(* Logix 5000 project; controller reports 1756-L63 rev 20.11; software revision 20.04; part 18 of 52 *)

        [994].time.Day := 13, [994].time.Hour := 3, [994].time.Minute := 14, [994].time.Second := 59, [995].log_data[0].min := 1.0, [995].log_data[0].max := 1.0, [995].log_data[0].total := 300.0, [995].log_data[0].time := 300.0, [995].log_data[0].minminute := 15, [995].log_data[0].maxminute := 15, [995].log_data[0].valid := 1, [995].log_data[1].valid := 1, [995].log_data[2].valid := 1, [995].log_data[3].valid := 1, [995].log_data[4].valid := 1, [995].log_data[5].valid := 1, [995].log_data[6].valid := 1, [995].log_data[7].valid := 1, [995].log_data[8].valid := 1, [995].log_data[9].valid := 1, [995].log_data[10].valid := 1, [995].log_data[11].valid := 1, [995].log_data[12].valid := 1, [995].log_data[13].valid := 1, [995].log_data[14].valid := 1, [995].log_data[15].valid := 1, [995].log_data[16].valid := 1, [995].log_data[17].valid := 1, [995].log_data[18].valid := 1, [995].log_data[19].valid := 1, [995].time.Year := 2023, [995].time.Month := 1, [995].time.Day := 13, [995].time.Hour := 3, [995].time.Minute := 19, [995].time.Second := 59, [996].log_data[0].min := 1.0, [996].log_data[0].max := 1.0, [996].log_data[0].total := 300.0, [996].log_data[0].time := 300.0, [996].log_data[0].minminute := 20, [996].log_data[0].maxminute := 20, [996].log_data[0].valid := 1, [996].log_data[1].valid := 1, [996].log_data[2].valid := 1, [996].log_data[3].valid := 1, [996].log_data[4].valid := 1, [996].log_data[5].valid := 1, [996].log_data[6].valid := 1, [996].log_data[7].valid := 1, [996].log_data[8].valid := 1, [996].log_data[9].valid := 1, [996].log_data[10].valid := 1, [996].log_data[11].valid := 1, [996].log_data[12].valid := 1, [996].log_data[13].valid := 1, [996].log_data[14].valid := 1, [996].log_data[15].valid := 1, [996].log_data[16].valid := 1, [996].log_data[17].valid := 1,
        [996].log_data[18].valid := 1, [996].log_data[19].valid := 1, [996].time.Year := 2023, [996].time.Month := 1, [996].time.Day := 13, [996].time.Hour := 3, [996].time.Minute := 24, [996].time.Second := 59, [997].log_data[0].min := 1.0, [997].log_data[0].max := 1.0, [997].log_data[0].total := 300.0, [997].log_data[0].time := 300.0, [997].log_data[0].minminute := 25, [997].log_data[0].maxminute := 25, [997].log_data[0].valid := 1, [997].log_data[1].valid := 1, [997].log_data[2].valid := 1, [997].log_data[3].valid := 1, [997].log_data[4].valid := 1, [997].log_data[5].valid := 1, [997].log_data[6].valid := 1, [997].log_data[7].valid := 1, [997].log_data[8].valid := 1, [997].log_data[9].valid := 1, [997].log_data[10].valid := 1, [997].log_data[11].valid := 1, [997].log_data[12].valid := 1, [997].log_data[13].valid := 1, [997].log_data[14].valid := 1, [997].log_data[15].valid := 1, [997].log_data[16].valid := 1, [997].log_data[17].valid := 1, [997].log_data[18].valid := 1, [997].log_data[19].valid := 1, [997].time.Year := 2023, [997].time.Month := 1, [997].time.Day := 13, [997].time.Hour := 3, [997].time.Minute := 29, [997].time.Second := 59, [998].log_data[0].min := 1.0, [998].log_data[0].max := 1.0, [998].log_data[0].total := 300.0, [998].log_data[0].time := 300.0, [998].log_data[0].minminute := 30, [998].log_data[0].maxminute := 30, [998].log_data[0].valid := 1, [998].log_data[1].valid := 1, [998].log_data[2].valid := 1, [998].log_data[3].valid := 1, [998].log_data[4].valid := 1, [998].log_data[5].valid := 1, [998].log_data[6].valid := 1, [998].log_data[7].valid := 1, [998].log_data[8].valid := 1, [998].log_data[9].valid := 1, [998].log_data[10].valid := 1, [998].log_data[11].valid := 1, [998].log_data[12].valid := 1, [998].log_data[13].valid := 1,
        [998].log_data[14].valid := 1, [998].log_data[15].valid := 1, [998].log_data[16].valid := 1, [998].log_data[17].valid := 1, [998].log_data[18].valid := 1, [998].log_data[19].valid := 1, [998].time.Year := 2023, [998].time.Month := 1, [998].time.Day := 13, [998].time.Hour := 3, [998].time.Minute := 34, [998].time.Second := 59, [999].log_data[0].min := 1.0, [999].log_data[0].max := 1.0, [999].log_data[0].total := 300.0, [999].log_data[0].time := 300.0, [999].log_data[0].minminute := 35, [999].log_data[0].maxminute := 35, [999].log_data[0].valid := 1, [999].log_data[1].valid := 1, [999].log_data[2].valid := 1, [999].log_data[3].valid := 1, [999].log_data[4].valid := 1, [999].log_data[5].valid := 1, [999].log_data[6].valid := 1, [999].log_data[7].valid := 1, [999].log_data[8].valid := 1, [999].log_data[9].valid := 1, [999].log_data[10].valid := 1, [999].log_data[11].valid := 1, [999].log_data[12].valid := 1, [999].log_data[13].valid := 1, [999].log_data[14].valid := 1, [999].log_data[15].valid := 1, [999].log_data[16].valid := 1, [999].log_data[17].valid := 1, [999].log_data[18].valid := 1, [999].log_data[19].valid := 1, [999].time.Year := 2023, [999].time.Month := 1, [999].time.Day := 13, [999].time.Hour := 3, [999].time.Minute := 39, [999].time.Second := 59, [1000].log_data[0].min := 1.0, [1000].log_data[0].max := 1.0, [1000].log_data[0].total := 300.0, [1000].log_data[0].time := 300.0, [1000].log_data[0].minminute := 40, [1000].log_data[0].maxminute := 40, [1000].log_data[0].valid := 1, [1000].log_data[1].valid := 1, [1000].log_data[2].valid := 1, [1000].log_data[3].valid := 1, [1000].log_data[4].valid := 1, [1000].log_data[5].valid := 1, [1000].log_data[6].valid := 1, [1000].log_data[7].valid := 1, [1000].log_data[8].valid := 1, [1000].log_data[9].valid := 1,
        [1000].log_data[10].valid := 1, [1000].log_data[11].valid := 1, [1000].log_data[12].valid := 1, [1000].log_data[13].valid := 1, [1000].log_data[14].valid := 1, [1000].log_data[15].valid := 1, [1000].log_data[16].valid := 1, [1000].log_data[17].valid := 1, [1000].log_data[18].valid := 1, [1000].log_data[19].valid := 1, [1000].time.Year := 2023, [1000].time.Month := 1, [1000].time.Day := 13, [1000].time.Hour := 3, [1000].time.Minute := 44, [1000].time.Second := 59, [1001].log_data[0].min := 1.0, [1001].log_data[0].max := 1.0, [1001].log_data[0].total := 300.0, [1001].log_data[0].time := 300.0, [1001].log_data[0].minminute := 45, [1001].log_data[0].maxminute := 45, [1001].log_data[0].valid := 1, [1001].log_data[1].valid := 1, [1001].log_data[2].valid := 1, [1001].log_data[3].valid := 1, [1001].log_data[4].valid := 1, [1001].log_data[5].valid := 1, [1001].log_data[6].valid := 1, [1001].log_data[7].valid := 1, [1001].log_data[8].valid := 1, [1001].log_data[9].valid := 1, [1001].log_data[10].valid := 1, [1001].log_data[11].valid := 1, [1001].log_data[12].valid := 1, [1001].log_data[13].valid := 1, [1001].log_data[14].valid := 1, [1001].log_data[15].valid := 1, [1001].log_data[16].valid := 1, [1001].log_data[17].valid := 1, [1001].log_data[18].valid := 1, [1001].log_data[19].valid := 1, [1001].time.Year := 2023, [1001].time.Month := 1, [1001].time.Day := 13, [1001].time.Hour := 3, [1001].time.Minute := 49, [1001].time.Second := 59, [1002].log_data[0].min := 1.0, [1002].log_data[0].max := 1.0, [1002].log_data[0].total := 300.0, [1002].log_data[0].time := 300.0, [1002].log_data[0].minminute := 50, [1002].log_data[0].maxminute := 50, [1002].log_data[0].valid := 1, [1002].log_data[1].valid := 1, [1002].log_data[2].valid := 1, [1002].log_data[3].valid := 1, [1002].log_data[4].valid := 1, [1002].log_data[5].valid := 1,
        [1002].log_data[6].valid := 1, [1002].log_data[7].valid := 1, [1002].log_data[8].valid := 1, [1002].log_data[9].valid := 1, [1002].log_data[10].valid := 1, [1002].log_data[11].valid := 1, [1002].log_data[12].valid := 1, [1002].log_data[13].valid := 1, [1002].log_data[14].valid := 1, [1002].log_data[15].valid := 1, [1002].log_data[16].valid := 1, [1002].log_data[17].valid := 1, [1002].log_data[18].valid := 1, [1002].log_data[19].valid := 1, [1002].time.Year := 2023, [1002].time.Month := 1, [1002].time.Day := 13, [1002].time.Hour := 3, [1002].time.Minute := 54, [1002].time.Second := 59, [1003].log_data[0].min := 1.0, [1003].log_data[0].max := 1.0, [1003].log_data[0].total := 300.0, [1003].log_data[0].time := 300.0, [1003].log_data[0].minminute := 55, [1003].log_data[0].maxminute := 55, [1003].log_data[0].valid := 1, [1003].log_data[1].valid := 1, [1003].log_data[2].valid := 1, [1003].log_data[3].valid := 1, [1003].log_data[4].valid := 1, [1003].log_data[5].valid := 1, [1003].log_data[6].valid := 1, [1003].log_data[7].valid := 1, [1003].log_data[8].valid := 1, [1003].log_data[9].valid := 1, [1003].log_data[10].valid := 1, [1003].log_data[11].valid := 1, [1003].log_data[12].valid := 1, [1003].log_data[13].valid := 1, [1003].log_data[14].valid := 1, [1003].log_data[15].valid := 1, [1003].log_data[16].valid := 1, [1003].log_data[17].valid := 1, [1003].log_data[18].valid := 1, [1003].log_data[19].valid := 1, [1003].time.Year := 2023, [1003].time.Month := 1, [1003].time.Day := 13, [1003].time.Hour := 3, [1003].time.Minute := 59, [1003].time.Second := 59, [1004].log_data[0].min := 1.0, [1004].log_data[0].max := 1.0, [1004].log_data[0].total := 300.0, [1004].log_data[0].time := 300.0, [1004].log_data[0].valid := 1, [1004].log_data[1].valid := 1, [1004].log_data[2].valid := 1, [1004].log_data[3].valid := 1,
        [1004].log_data[4].valid := 1, [1004].log_data[5].valid := 1, [1004].log_data[6].valid := 1, [1004].log_data[7].valid := 1, [1004].log_data[8].valid := 1, [1004].log_data[9].valid := 1, [1004].log_data[10].valid := 1, [1004].log_data[11].valid := 1, [1004].log_data[12].valid := 1, [1004].log_data[13].valid := 1, [1004].log_data[14].valid := 1, [1004].log_data[15].valid := 1, [1004].log_data[16].valid := 1, [1004].log_data[17].valid := 1, [1004].log_data[18].valid := 1, [1004].log_data[19].valid := 1, [1004].time.Year := 2023, [1004].time.Month := 1, [1004].time.Day := 13, [1004].time.Hour := 4, [1004].time.Minute := 4, [1004].time.Second := 59, [1005].log_data[0].min := 1.0, [1005].log_data[0].max := 1.0, [1005].log_data[0].total := 300.0, [1005].log_data[0].time := 300.0, [1005].log_data[0].minminute := 5, [1005].log_data[0].maxminute := 5, [1005].log_data[0].valid := 1, [1005].log_data[1].valid := 1, [1005].log_data[2].valid := 1, [1005].log_data[3].valid := 1, [1005].log_data[4].valid := 1, [1005].log_data[5].valid := 1, [1005].log_data[6].valid := 1, [1005].log_data[7].valid := 1, [1005].log_data[8].valid := 1, [1005].log_data[9].valid := 1, [1005].log_data[10].valid := 1, [1005].log_data[11].valid := 1, [1005].log_data[12].valid := 1, [1005].log_data[13].valid := 1, [1005].log_data[14].valid := 1, [1005].log_data[15].valid := 1, [1005].log_data[16].valid := 1, [1005].log_data[17].valid := 1, [1005].log_data[18].valid := 1, [1005].log_data[19].valid := 1, [1005].time.Year := 2023, [1005].time.Month := 1, [1005].time.Day := 13, [1005].time.Hour := 4, [1005].time.Minute := 9, [1005].time.Second := 59, [1006].log_data[0].min := 1.0, [1006].log_data[0].max := 1.0, [1006].log_data[0].total := 300.0, [1006].log_data[0].time := 300.0, [1006].log_data[0].minminute := 10, [1006].log_data[0].maxminute := 10,
        [1006].log_data[0].valid := 1, [1006].log_data[1].valid := 1, [1006].log_data[2].valid := 1, [1006].log_data[3].valid := 1, [1006].log_data[4].valid := 1, [1006].log_data[5].valid := 1, [1006].log_data[6].valid := 1, [1006].log_data[7].valid := 1, [1006].log_data[8].valid := 1, [1006].log_data[9].valid := 1, [1006].log_data[10].valid := 1, [1006].log_data[11].valid := 1, [1006].log_data[12].valid := 1, [1006].log_data[13].valid := 1, [1006].log_data[14].valid := 1, [1006].log_data[15].valid := 1, [1006].log_data[16].valid := 1, [1006].log_data[17].valid := 1, [1006].log_data[18].valid := 1, [1006].log_data[19].valid := 1, [1006].time.Year := 2023, [1006].time.Month := 1, [1006].time.Day := 13, [1006].time.Hour := 4, [1006].time.Minute := 14, [1006].time.Second := 59, [1007].log_data[0].min := 1.0, [1007].log_data[0].max := 1.0, [1007].log_data[0].total := 300.0, [1007].log_data[0].time := 300.0, [1007].log_data[0].minminute := 15, [1007].log_data[0].maxminute := 15, [1007].log_data[0].valid := 1, [1007].log_data[1].valid := 1, [1007].log_data[2].valid := 1, [1007].log_data[3].valid := 1, [1007].log_data[4].valid := 1, [1007].log_data[5].valid := 1, [1007].log_data[6].valid := 1, [1007].log_data[7].valid := 1, [1007].log_data[8].valid := 1, [1007].log_data[9].valid := 1, [1007].log_data[10].valid := 1, [1007].log_data[11].valid := 1, [1007].log_data[12].valid := 1, [1007].log_data[13].valid := 1, [1007].log_data[14].valid := 1, [1007].log_data[15].valid := 1, [1007].log_data[16].valid := 1, [1007].log_data[17].valid := 1, [1007].log_data[18].valid := 1, [1007].log_data[19].valid := 1, [1007].time.Year := 2023, [1007].time.Month := 1, [1007].time.Day := 13, [1007].time.Hour := 4, [1007].time.Minute := 19, [1007].time.Second := 59, [1008].log_data[0].min := 1.0, [1008].log_data[0].max := 1.0,
        [1008].log_data[0].total := 300.0, [1008].log_data[0].time := 300.0, [1008].log_data[0].minminute := 20, [1008].log_data[0].maxminute := 20, [1008].log_data[0].valid := 1, [1008].log_data[1].valid := 1, [1008].log_data[2].valid := 1, [1008].log_data[3].valid := 1, [1008].log_data[4].valid := 1, [1008].log_data[5].valid := 1, [1008].log_data[6].valid := 1, [1008].log_data[7].valid := 1, [1008].log_data[8].valid := 1, [1008].log_data[9].valid := 1, [1008].log_data[10].valid := 1, [1008].log_data[11].valid := 1, [1008].log_data[12].valid := 1, [1008].log_data[13].valid := 1, [1008].log_data[14].valid := 1, [1008].log_data[15].valid := 1, [1008].log_data[16].valid := 1, [1008].log_data[17].valid := 1, [1008].log_data[18].valid := 1, [1008].log_data[19].valid := 1, [1008].time.Year := 2023, [1008].time.Month := 1, [1008].time.Day := 13, [1008].time.Hour := 4, [1008].time.Minute := 24, [1008].time.Second := 59, [1009].log_data[0].min := 1.0, [1009].log_data[0].max := 1.0, [1009].log_data[0].total := 300.0, [1009].log_data[0].time := 300.0, [1009].log_data[0].minminute := 25, [1009].log_data[0].maxminute := 25, [1009].log_data[0].valid := 1, [1009].log_data[1].valid := 1, [1009].log_data[2].valid := 1, [1009].log_data[3].valid := 1, [1009].log_data[4].valid := 1, [1009].log_data[5].valid := 1, [1009].log_data[6].valid := 1, [1009].log_data[7].valid := 1, [1009].log_data[8].valid := 1, [1009].log_data[9].valid := 1, [1009].log_data[10].valid := 1, [1009].log_data[11].valid := 1, [1009].log_data[12].valid := 1, [1009].log_data[13].valid := 1, [1009].log_data[14].valid := 1, [1009].log_data[15].valid := 1, [1009].log_data[16].valid := 1, [1009].log_data[17].valid := 1, [1009].log_data[18].valid := 1, [1009].log_data[19].valid := 1, [1009].time.Year := 2023, [1009].time.Month := 1, [1009].time.Day := 13, [1009].time.Hour := 4,
        [1009].time.Minute := 29, [1009].time.Second := 59, [1010].log_data[0].min := 1.0, [1010].log_data[0].max := 1.0, [1010].log_data[0].total := 300.0, [1010].log_data[0].time := 300.0, [1010].log_data[0].minminute := 30, [1010].log_data[0].maxminute := 30, [1010].log_data[0].valid := 1, [1010].log_data[1].valid := 1, [1010].log_data[2].valid := 1, [1010].log_data[3].valid := 1, [1010].log_data[4].valid := 1, [1010].log_data[5].valid := 1, [1010].log_data[6].valid := 1, [1010].log_data[7].valid := 1, [1010].log_data[8].valid := 1, [1010].log_data[9].valid := 1, [1010].log_data[10].valid := 1, [1010].log_data[11].valid := 1, [1010].log_data[12].valid := 1, [1010].log_data[13].valid := 1, [1010].log_data[14].valid := 1, [1010].log_data[15].valid := 1, [1010].log_data[16].valid := 1, [1010].log_data[17].valid := 1, [1010].log_data[18].valid := 1, [1010].log_data[19].valid := 1, [1010].time.Year := 2023, [1010].time.Month := 1, [1010].time.Day := 13, [1010].time.Hour := 4, [1010].time.Minute := 34, [1010].time.Second := 59, [1011].log_data[0].min := 1.0, [1011].log_data[0].max := 1.0, [1011].log_data[0].total := 300.0, [1011].log_data[0].time := 300.0, [1011].log_data[0].minminute := 35, [1011].log_data[0].maxminute := 35, [1011].log_data[0].valid := 1, [1011].log_data[1].valid := 1, [1011].log_data[2].valid := 1, [1011].log_data[3].valid := 1, [1011].log_data[4].valid := 1, [1011].log_data[5].valid := 1, [1011].log_data[6].valid := 1, [1011].log_data[7].valid := 1, [1011].log_data[8].valid := 1, [1011].log_data[9].valid := 1, [1011].log_data[10].valid := 1, [1011].log_data[11].valid := 1, [1011].log_data[12].valid := 1, [1011].log_data[13].valid := 1, [1011].log_data[14].valid := 1, [1011].log_data[15].valid := 1, [1011].log_data[16].valid := 1, [1011].log_data[17].valid := 1, [1011].log_data[18].valid := 1, [1011].log_data[19].valid := 1,
        [1011].time.Year := 2023, [1011].time.Month := 1, [1011].time.Day := 13, [1011].time.Hour := 4, [1011].time.Minute := 39, [1011].time.Second := 59, [1012].log_data[0].min := 1.0, [1012].log_data[0].max := 1.0, [1012].log_data[0].total := 300.0, [1012].log_data[0].time := 300.0, [1012].log_data[0].minminute := 40, [1012].log_data[0].maxminute := 40, [1012].log_data[0].valid := 1, [1012].log_data[1].valid := 1, [1012].log_data[2].valid := 1, [1012].log_data[3].valid := 1, [1012].log_data[4].valid := 1, [1012].log_data[5].valid := 1, [1012].log_data[6].valid := 1, [1012].log_data[7].valid := 1, [1012].log_data[8].valid := 1, [1012].log_data[9].valid := 1, [1012].log_data[10].valid := 1, [1012].log_data[11].valid := 1, [1012].log_data[12].valid := 1, [1012].log_data[13].valid := 1, [1012].log_data[14].valid := 1, [1012].log_data[15].valid := 1, [1012].log_data[16].valid := 1, [1012].log_data[17].valid := 1, [1012].log_data[18].valid := 1, [1012].log_data[19].valid := 1, [1012].time.Year := 2023, [1012].time.Month := 1, [1012].time.Day := 13, [1012].time.Hour := 4, [1012].time.Minute := 44, [1012].time.Second := 59, [1013].log_data[0].min := 1.0, [1013].log_data[0].max := 1.0, [1013].log_data[0].total := 300.0, [1013].log_data[0].time := 300.0, [1013].log_data[0].minminute := 45, [1013].log_data[0].maxminute := 45, [1013].log_data[0].valid := 1, [1013].log_data[1].valid := 1, [1013].log_data[2].valid := 1, [1013].log_data[3].valid := 1, [1013].log_data[4].valid := 1, [1013].log_data[5].valid := 1, [1013].log_data[6].valid := 1, [1013].log_data[7].valid := 1, [1013].log_data[8].valid := 1, [1013].log_data[9].valid := 1, [1013].log_data[10].valid := 1, [1013].log_data[11].valid := 1, [1013].log_data[12].valid := 1, [1013].log_data[13].valid := 1, [1013].log_data[14].valid := 1, [1013].log_data[15].valid := 1,
        [1013].log_data[16].valid := 1, [1013].log_data[17].valid := 1, [1013].log_data[18].valid := 1, [1013].log_data[19].valid := 1, [1013].time.Year := 2023, [1013].time.Month := 1, [1013].time.Day := 13, [1013].time.Hour := 4, [1013].time.Minute := 49, [1013].time.Second := 59, [1014].log_data[0].min := 1.0, [1014].log_data[0].max := 1.0, [1014].log_data[0].total := 300.0, [1014].log_data[0].time := 300.0, [1014].log_data[0].minminute := 50, [1014].log_data[0].maxminute := 50, [1014].log_data[0].valid := 1, [1014].log_data[1].valid := 1, [1014].log_data[2].valid := 1, [1014].log_data[3].valid := 1, [1014].log_data[4].valid := 1, [1014].log_data[5].valid := 1, [1014].log_data[6].valid := 1, [1014].log_data[7].valid := 1, [1014].log_data[8].valid := 1, [1014].log_data[9].valid := 1, [1014].log_data[10].valid := 1, [1014].log_data[11].valid := 1, [1014].log_data[12].valid := 1, [1014].log_data[13].valid := 1, [1014].log_data[14].valid := 1, [1014].log_data[15].valid := 1, [1014].log_data[16].valid := 1, [1014].log_data[17].valid := 1, [1014].log_data[18].valid := 1, [1014].log_data[19].valid := 1, [1014].time.Year := 2023, [1014].time.Month := 1, [1014].time.Day := 13, [1014].time.Hour := 4, [1014].time.Minute := 54, [1014].time.Second := 59, [1015].log_data[0].min := 1.0, [1015].log_data[0].max := 1.0, [1015].log_data[0].total := 300.0, [1015].log_data[0].time := 300.0, [1015].log_data[0].minminute := 55, [1015].log_data[0].maxminute := 55, [1015].log_data[0].valid := 1, [1015].log_data[1].valid := 1, [1015].log_data[2].valid := 1, [1015].log_data[3].valid := 1, [1015].log_data[4].valid := 1, [1015].log_data[5].valid := 1, [1015].log_data[6].valid := 1, [1015].log_data[7].valid := 1, [1015].log_data[8].valid := 1, [1015].log_data[9].valid := 1, [1015].log_data[10].valid := 1, [1015].log_data[11].valid := 1,
        [1015].log_data[12].valid := 1, [1015].log_data[13].valid := 1, [1015].log_data[14].valid := 1, [1015].log_data[15].valid := 1, [1015].log_data[16].valid := 1, [1015].log_data[17].valid := 1, [1015].log_data[18].valid := 1, [1015].log_data[19].valid := 1, [1015].time.Year := 2023, [1015].time.Month := 1, [1015].time.Day := 13, [1015].time.Hour := 4, [1015].time.Minute := 59, [1015].time.Second := 59, [1016].log_data[0].min := 1.0, [1016].log_data[0].max := 1.0, [1016].log_data[0].total := 300.0, [1016].log_data[0].time := 300.0, [1016].log_data[0].valid := 1, [1016].log_data[1].valid := 1, [1016].log_data[2].valid := 1, [1016].log_data[3].valid := 1, [1016].log_data[4].valid := 1, [1016].log_data[5].valid := 1, [1016].log_data[6].valid := 1, [1016].log_data[7].valid := 1, [1016].log_data[8].valid := 1, [1016].log_data[9].valid := 1, [1016].log_data[10].valid := 1, [1016].log_data[11].valid := 1, [1016].log_data[12].valid := 1, [1016].log_data[13].valid := 1, [1016].log_data[14].valid := 1, [1016].log_data[15].valid := 1, [1016].log_data[16].valid := 1, [1016].log_data[17].valid := 1, [1016].log_data[18].valid := 1, [1016].log_data[19].valid := 1, [1016].time.Year := 2023, [1016].time.Month := 1, [1016].time.Day := 13, [1016].time.Hour := 5, [1016].time.Minute := 4, [1016].time.Second := 59, [1017].log_data[0].min := 1.0, [1017].log_data[0].max := 1.0, [1017].log_data[0].total := 300.0, [1017].log_data[0].time := 300.0, [1017].log_data[0].minminute := 5, [1017].log_data[0].maxminute := 5, [1017].log_data[0].valid := 1, [1017].log_data[1].valid := 1, [1017].log_data[2].valid := 1, [1017].log_data[3].valid := 1, [1017].log_data[4].valid := 1, [1017].log_data[5].valid := 1, [1017].log_data[6].valid := 1, [1017].log_data[7].valid := 1, [1017].log_data[8].valid := 1, [1017].log_data[9].valid := 1,
        [1017].log_data[10].valid := 1, [1017].log_data[11].valid := 1, [1017].log_data[12].valid := 1, [1017].log_data[13].valid := 1, [1017].log_data[14].valid := 1, [1017].log_data[15].valid := 1, [1017].log_data[16].valid := 1, [1017].log_data[17].valid := 1, [1017].log_data[18].valid := 1, [1017].log_data[19].valid := 1, [1017].time.Year := 2023, [1017].time.Month := 1, [1017].time.Day := 13, [1017].time.Hour := 5, [1017].time.Minute := 9, [1017].time.Second := 59, [1018].log_data[0].min := 1.0, [1018].log_data[0].max := 1.0, [1018].log_data[0].total := 300.0, [1018].log_data[0].time := 300.0, [1018].log_data[0].minminute := 10, [1018].log_data[0].maxminute := 10, [1018].log_data[0].valid := 1, [1018].log_data[1].valid := 1, [1018].log_data[2].valid := 1, [1018].log_data[3].valid := 1, [1018].log_data[4].valid := 1, [1018].log_data[5].valid := 1, [1018].log_data[6].valid := 1, [1018].log_data[7].valid := 1, [1018].log_data[8].valid := 1, [1018].log_data[9].valid := 1, [1018].log_data[10].valid := 1, [1018].log_data[11].valid := 1, [1018].log_data[12].valid := 1, [1018].log_data[13].valid := 1, [1018].log_data[14].valid := 1, [1018].log_data[15].valid := 1, [1018].log_data[16].valid := 1, [1018].log_data[17].valid := 1, [1018].log_data[18].valid := 1, [1018].log_data[19].valid := 1, [1018].time.Year := 2023, [1018].time.Month := 1, [1018].time.Day := 13, [1018].time.Hour := 5, [1018].time.Minute := 14, [1018].time.Second := 59, [1019].log_data[0].min := 1.0, [1019].log_data[0].max := 1.0, [1019].log_data[0].total := 300.0, [1019].log_data[0].time := 300.0, [1019].log_data[0].minminute := 15, [1019].log_data[0].maxminute := 15, [1019].log_data[0].valid := 1, [1019].log_data[1].valid := 1, [1019].log_data[2].valid := 1, [1019].log_data[3].valid := 1, [1019].log_data[4].valid := 1, [1019].log_data[5].valid := 1,
        [1019].log_data[6].valid := 1, [1019].log_data[7].valid := 1, [1019].log_data[8].valid := 1, [1019].log_data[9].valid := 1, [1019].log_data[10].valid := 1, [1019].log_data[11].valid := 1, [1019].log_data[12].valid := 1, [1019].log_data[13].valid := 1, [1019].log_data[14].valid := 1, [1019].log_data[15].valid := 1, [1019].log_data[16].valid := 1, [1019].log_data[17].valid := 1, [1019].log_data[18].valid := 1, [1019].log_data[19].valid := 1, [1019].time.Year := 2023, [1019].time.Month := 1, [1019].time.Day := 13, [1019].time.Hour := 5, [1019].time.Minute := 19, [1019].time.Second := 59, [1020].log_data[0].min := 1.0, [1020].log_data[0].max := 1.0, [1020].log_data[0].total := 300.0, [1020].log_data[0].time := 300.0, [1020].log_data[0].minminute := 20, [1020].log_data[0].maxminute := 20, [1020].log_data[0].valid := 1, [1020].log_data[1].valid := 1, [1020].log_data[2].valid := 1, [1020].log_data[3].valid := 1, [1020].log_data[4].valid := 1, [1020].log_data[5].valid := 1, [1020].log_data[6].valid := 1, [1020].log_data[7].valid := 1, [1020].log_data[8].valid := 1, [1020].log_data[9].valid := 1, [1020].log_data[10].valid := 1, [1020].log_data[11].valid := 1, [1020].log_data[12].valid := 1, [1020].log_data[13].valid := 1, [1020].log_data[14].valid := 1, [1020].log_data[15].valid := 1, [1020].log_data[16].valid := 1, [1020].log_data[17].valid := 1, [1020].log_data[18].valid := 1, [1020].log_data[19].valid := 1, [1020].time.Year := 2023, [1020].time.Month := 1, [1020].time.Day := 13, [1020].time.Hour := 5, [1020].time.Minute := 24, [1020].time.Second := 59, [1021].log_data[0].min := 1.0, [1021].log_data[0].max := 1.0, [1021].log_data[0].total := 300.0, [1021].log_data[0].time := 300.0, [1021].log_data[0].minminute := 25, [1021].log_data[0].maxminute := 25, [1021].log_data[0].valid := 1, [1021].log_data[1].valid := 1,
        [1021].log_data[2].valid := 1, [1021].log_data[3].valid := 1, [1021].log_data[4].valid := 1, [1021].log_data[5].valid := 1, [1021].log_data[6].valid := 1, [1021].log_data[7].valid := 1, [1021].log_data[8].valid := 1, [1021].log_data[9].valid := 1, [1021].log_data[10].valid := 1, [1021].log_data[11].valid := 1, [1021].log_data[12].valid := 1, [1021].log_data[13].valid := 1, [1021].log_data[14].valid := 1, [1021].log_data[15].valid := 1, [1021].log_data[16].valid := 1, [1021].log_data[17].valid := 1, [1021].log_data[18].valid := 1, [1021].log_data[19].valid := 1, [1021].time.Year := 2023, [1021].time.Month := 1, [1021].time.Day := 13, [1021].time.Hour := 5, [1021].time.Minute := 29, [1021].time.Second := 59, [1022].log_data[0].min := 1.0, [1022].log_data[0].max := 1.0, [1022].log_data[0].total := 300.0, [1022].log_data[0].time := 300.0, [1022].log_data[0].minminute := 30, [1022].log_data[0].maxminute := 30, [1022].log_data[0].valid := 1, [1022].log_data[1].valid := 1, [1022].log_data[2].valid := 1, [1022].log_data[3].valid := 1, [1022].log_data[4].valid := 1, [1022].log_data[5].valid := 1, [1022].log_data[6].valid := 1, [1022].log_data[7].valid := 1, [1022].log_data[8].valid := 1, [1022].log_data[9].valid := 1, [1022].log_data[10].valid := 1, [1022].log_data[11].valid := 1, [1022].log_data[12].valid := 1, [1022].log_data[13].valid := 1, [1022].log_data[14].valid := 1, [1022].log_data[15].valid := 1, [1022].log_data[16].valid := 1, [1022].log_data[17].valid := 1, [1022].log_data[18].valid := 1, [1022].log_data[19].valid := 1, [1022].time.Year := 2023, [1022].time.Month := 1, [1022].time.Day := 13, [1022].time.Hour := 5, [1022].time.Minute := 34, [1022].time.Second := 59, [1023].log_data[0].min := 1.0, [1023].log_data[0].max := 1.0, [1023].log_data[0].total := 300.0, [1023].log_data[0].time := 300.0,
        [1023].log_data[0].minminute := 35, [1023].log_data[0].maxminute := 35, [1023].log_data[0].valid := 1, [1023].log_data[1].valid := 1, [1023].log_data[2].valid := 1, [1023].log_data[3].valid := 1, [1023].log_data[4].valid := 1, [1023].log_data[5].valid := 1, [1023].log_data[6].valid := 1, [1023].log_data[7].valid := 1, [1023].log_data[8].valid := 1, [1023].log_data[9].valid := 1, [1023].log_data[10].valid := 1, [1023].log_data[11].valid := 1, [1023].log_data[12].valid := 1, [1023].log_data[13].valid := 1, [1023].log_data[14].valid := 1, [1023].log_data[15].valid := 1, [1023].log_data[16].valid := 1, [1023].log_data[17].valid := 1, [1023].log_data[18].valid := 1, [1023].log_data[19].valid := 1, [1023].time.Year := 2023, [1023].time.Month := 1, [1023].time.Day := 13, [1023].time.Hour := 5, [1023].time.Minute := 39, [1023].time.Second := 59, [1024].log_data[0].min := 1.0, [1024].log_data[0].max := 1.0, [1024].log_data[0].total := 300.0, [1024].log_data[0].time := 300.0, [1024].log_data[0].minminute := 40, [1024].log_data[0].maxminute := 40, [1024].log_data[0].valid := 1, [1024].log_data[1].valid := 1, [1024].log_data[2].valid := 1, [1024].log_data[3].valid := 1, [1024].log_data[4].valid := 1, [1024].log_data[5].valid := 1, [1024].log_data[6].valid := 1, [1024].log_data[7].valid := 1, [1024].log_data[8].valid := 1, [1024].log_data[9].valid := 1, [1024].log_data[10].valid := 1, [1024].log_data[11].valid := 1, [1024].log_data[12].valid := 1, [1024].log_data[13].valid := 1, [1024].log_data[14].valid := 1, [1024].log_data[15].valid := 1, [1024].log_data[16].valid := 1, [1024].log_data[17].valid := 1, [1024].log_data[18].valid := 1, [1024].log_data[19].valid := 1, [1024].time.Year := 2023, [1024].time.Month := 1, [1024].time.Day := 13, [1024].time.Hour := 5, [1024].time.Minute := 44, [1024].time.Second := 59,
        [1025].log_data[0].min := 1.0, [1025].log_data[0].max := 1.0, [1025].log_data[0].total := 300.0, [1025].log_data[0].time := 300.0, [1025].log_data[0].minminute := 45, [1025].log_data[0].maxminute := 45, [1025].log_data[0].valid := 1, [1025].log_data[1].valid := 1, [1025].log_data[2].valid := 1, [1025].log_data[3].valid := 1, [1025].log_data[4].valid := 1, [1025].log_data[5].valid := 1, [1025].log_data[6].valid := 1, [1025].log_data[7].valid := 1, [1025].log_data[8].valid := 1, [1025].log_data[9].valid := 1, [1025].log_data[10].valid := 1, [1025].log_data[11].valid := 1, [1025].log_data[12].valid := 1, [1025].log_data[13].valid := 1, [1025].log_data[14].valid := 1, [1025].log_data[15].valid := 1, [1025].log_data[16].valid := 1, [1025].log_data[17].valid := 1, [1025].log_data[18].valid := 1, [1025].log_data[19].valid := 1, [1025].time.Year := 2023, [1025].time.Month := 1, [1025].time.Day := 13, [1025].time.Hour := 5, [1025].time.Minute := 49, [1025].time.Second := 59, [1026].log_data[0].min := 1.0, [1026].log_data[0].max := 1.0, [1026].log_data[0].total := 300.0, [1026].log_data[0].time := 300.0, [1026].log_data[0].minminute := 50, [1026].log_data[0].maxminute := 50, [1026].log_data[0].valid := 1, [1026].log_data[1].valid := 1, [1026].log_data[2].valid := 1, [1026].log_data[3].valid := 1, [1026].log_data[4].valid := 1, [1026].log_data[5].valid := 1, [1026].log_data[6].valid := 1, [1026].log_data[7].valid := 1, [1026].log_data[8].valid := 1, [1026].log_data[9].valid := 1, [1026].log_data[10].valid := 1, [1026].log_data[11].valid := 1, [1026].log_data[12].valid := 1, [1026].log_data[13].valid := 1, [1026].log_data[14].valid := 1, [1026].log_data[15].valid := 1, [1026].log_data[16].valid := 1, [1026].log_data[17].valid := 1, [1026].log_data[18].valid := 1, [1026].log_data[19].valid := 1, [1026].time.Year := 2023, [1026].time.Month := 1,
        [1026].time.Day := 13, [1026].time.Hour := 5, [1026].time.Minute := 54, [1026].time.Second := 59, [1027].log_data[0].min := 1.0, [1027].log_data[0].max := 1.0, [1027].log_data[0].total := 300.0, [1027].log_data[0].time := 300.0, [1027].log_data[0].minminute := 55, [1027].log_data[0].maxminute := 55, [1027].log_data[0].valid := 1, [1027].log_data[1].valid := 1, [1027].log_data[2].valid := 1, [1027].log_data[3].valid := 1, [1027].log_data[4].valid := 1, [1027].log_data[5].valid := 1, [1027].log_data[6].valid := 1, [1027].log_data[7].valid := 1, [1027].log_data[8].valid := 1, [1027].log_data[9].valid := 1, [1027].log_data[10].valid := 1, [1027].log_data[11].valid := 1, [1027].log_data[12].valid := 1, [1027].log_data[13].valid := 1, [1027].log_data[14].valid := 1, [1027].log_data[15].valid := 1, [1027].log_data[16].valid := 1, [1027].log_data[17].valid := 1, [1027].log_data[18].valid := 1, [1027].log_data[19].valid := 1, [1027].time.Year := 2023, [1027].time.Month := 1, [1027].time.Day := 13, [1027].time.Hour := 5, [1027].time.Minute := 59, [1027].time.Second := 59, [1028].log_data[0].min := 1.0, [1028].log_data[0].max := 1.0, [1028].log_data[0].total := 300.0, [1028].log_data[0].time := 300.0, [1028].log_data[0].valid := 1, [1028].log_data[1].valid := 1, [1028].log_data[2].valid := 1, [1028].log_data[3].valid := 1, [1028].log_data[4].valid := 1, [1028].log_data[5].valid := 1, [1028].log_data[6].valid := 1, [1028].log_data[7].valid := 1, [1028].log_data[8].valid := 1, [1028].log_data[9].valid := 1, [1028].log_data[10].valid := 1, [1028].log_data[11].valid := 1, [1028].log_data[12].valid := 1, [1028].log_data[13].valid := 1, [1028].log_data[14].valid := 1, [1028].log_data[15].valid := 1, [1028].log_data[16].valid := 1, [1028].log_data[17].valid := 1, [1028].log_data[18].valid := 1, [1028].log_data[19].valid := 1,
        [1028].time.Year := 2023, [1028].time.Month := 1, [1028].time.Day := 13, [1028].time.Hour := 6, [1028].time.Minute := 4, [1028].time.Second := 59, [1029].log_data[0].min := 1.0, [1029].log_data[0].max := 1.0, [1029].log_data[0].total := 300.0, [1029].log_data[0].time := 300.0, [1029].log_data[0].minminute := 5, [1029].log_data[0].maxminute := 5, [1029].log_data[0].valid := 1, [1029].log_data[1].valid := 1, [1029].log_data[2].valid := 1, [1029].log_data[3].valid := 1, [1029].log_data[4].valid := 1, [1029].log_data[5].valid := 1, [1029].log_data[6].valid := 1, [1029].log_data[7].valid := 1, [1029].log_data[8].valid := 1, [1029].log_data[9].valid := 1, [1029].log_data[10].valid := 1, [1029].log_data[11].valid := 1, [1029].log_data[12].valid := 1, [1029].log_data[13].valid := 1, [1029].log_data[14].valid := 1, [1029].log_data[15].valid := 1, [1029].log_data[16].valid := 1, [1029].log_data[17].valid := 1, [1029].log_data[18].valid := 1, [1029].log_data[19].valid := 1, [1029].time.Year := 2023, [1029].time.Month := 1, [1029].time.Day := 13, [1029].time.Hour := 6, [1029].time.Minute := 9, [1029].time.Second := 59, [1030].log_data[0].min := 1.0, [1030].log_data[0].max := 1.0, [1030].log_data[0].total := 300.0, [1030].log_data[0].time := 300.0, [1030].log_data[0].minminute := 10, [1030].log_data[0].maxminute := 10, [1030].log_data[0].valid := 1, [1030].log_data[1].valid := 1, [1030].log_data[2].valid := 1, [1030].log_data[3].valid := 1, [1030].log_data[4].valid := 1, [1030].log_data[5].valid := 1, [1030].log_data[6].valid := 1, [1030].log_data[7].valid := 1, [1030].log_data[8].valid := 1, [1030].log_data[9].valid := 1, [1030].log_data[10].valid := 1, [1030].log_data[11].valid := 1, [1030].log_data[12].valid := 1, [1030].log_data[13].valid := 1, [1030].log_data[14].valid := 1, [1030].log_data[15].valid := 1,
        [1030].log_data[16].valid := 1, [1030].log_data[17].valid := 1, [1030].log_data[18].valid := 1, [1030].log_data[19].valid := 1, [1030].time.Year := 2023, [1030].time.Month := 1, [1030].time.Day := 13, [1030].time.Hour := 6, [1030].time.Minute := 14, [1030].time.Second := 59, [1031].log_data[0].min := 1.0, [1031].log_data[0].max := 1.0, [1031].log_data[0].total := 300.0, [1031].log_data[0].time := 300.0, [1031].log_data[0].minminute := 15, [1031].log_data[0].maxminute := 15, [1031].log_data[0].valid := 1, [1031].log_data[1].valid := 1, [1031].log_data[2].valid := 1, [1031].log_data[3].valid := 1, [1031].log_data[4].valid := 1, [1031].log_data[5].valid := 1, [1031].log_data[6].valid := 1, [1031].log_data[7].valid := 1, [1031].log_data[8].valid := 1, [1031].log_data[9].valid := 1, [1031].log_data[10].valid := 1, [1031].log_data[11].valid := 1, [1031].log_data[12].valid := 1, [1031].log_data[13].valid := 1, [1031].log_data[14].valid := 1, [1031].log_data[15].valid := 1, [1031].log_data[16].valid := 1, [1031].log_data[17].valid := 1, [1031].log_data[18].valid := 1, [1031].log_data[19].valid := 1, [1031].time.Year := 2023, [1031].time.Month := 1, [1031].time.Day := 13, [1031].time.Hour := 6, [1031].time.Minute := 19, [1031].time.Second := 59, [1032].log_data[0].min := 1.0, [1032].log_data[0].max := 1.0, [1032].log_data[0].total := 300.0, [1032].log_data[0].time := 300.0, [1032].log_data[0].minminute := 20, [1032].log_data[0].maxminute := 20, [1032].log_data[0].valid := 1, [1032].log_data[1].valid := 1, [1032].log_data[2].valid := 1, [1032].log_data[3].valid := 1, [1032].log_data[4].valid := 1, [1032].log_data[5].valid := 1, [1032].log_data[6].valid := 1, [1032].log_data[7].valid := 1, [1032].log_data[8].valid := 1, [1032].log_data[9].valid := 1, [1032].log_data[10].valid := 1, [1032].log_data[11].valid := 1,
        [1032].log_data[12].valid := 1, [1032].log_data[13].valid := 1, [1032].log_data[14].valid := 1, [1032].log_data[15].valid := 1, [1032].log_data[16].valid := 1, [1032].log_data[17].valid := 1, [1032].log_data[18].valid := 1, [1032].log_data[19].valid := 1, [1032].time.Year := 2023, [1032].time.Month := 1, [1032].time.Day := 13, [1032].time.Hour := 6, [1032].time.Minute := 24, [1032].time.Second := 59, [1033].log_data[0].min := 1.0, [1033].log_data[0].max := 1.0, [1033].log_data[0].total := 300.0, [1033].log_data[0].time := 300.0, [1033].log_data[0].minminute := 25, [1033].log_data[0].maxminute := 25, [1033].log_data[0].valid := 1, [1033].log_data[1].valid := 1, [1033].log_data[2].valid := 1, [1033].log_data[3].valid := 1, [1033].log_data[4].valid := 1, [1033].log_data[5].valid := 1, [1033].log_data[6].valid := 1, [1033].log_data[7].valid := 1, [1033].log_data[8].valid := 1, [1033].log_data[9].valid := 1, [1033].log_data[10].valid := 1, [1033].log_data[11].valid := 1, [1033].log_data[12].valid := 1, [1033].log_data[13].valid := 1, [1033].log_data[14].valid := 1, [1033].log_data[15].valid := 1, [1033].log_data[16].valid := 1, [1033].log_data[17].valid := 1, [1033].log_data[18].valid := 1, [1033].log_data[19].valid := 1, [1033].time.Year := 2023, [1033].time.Month := 1, [1033].time.Day := 13, [1033].time.Hour := 6, [1033].time.Minute := 29, [1033].time.Second := 59, [1034].log_data[0].min := 1.0, [1034].log_data[0].max := 1.0, [1034].log_data[0].total := 300.0, [1034].log_data[0].time := 300.0, [1034].log_data[0].minminute := 30, [1034].log_data[0].maxminute := 30, [1034].log_data[0].valid := 1, [1034].log_data[1].valid := 1, [1034].log_data[2].valid := 1, [1034].log_data[3].valid := 1, [1034].log_data[4].valid := 1, [1034].log_data[5].valid := 1, [1034].log_data[6].valid := 1, [1034].log_data[7].valid := 1,
        [1034].log_data[8].valid := 1, [1034].log_data[9].valid := 1, [1034].log_data[10].valid := 1, [1034].log_data[11].valid := 1, [1034].log_data[12].valid := 1, [1034].log_data[13].valid := 1, [1034].log_data[14].valid := 1, [1034].log_data[15].valid := 1, [1034].log_data[16].valid := 1, [1034].log_data[17].valid := 1, [1034].log_data[18].valid := 1, [1034].log_data[19].valid := 1, [1034].time.Year := 2023, [1034].time.Month := 1, [1034].time.Day := 13, [1034].time.Hour := 6, [1034].time.Minute := 34, [1034].time.Second := 59, [1035].log_data[0].min := 1.0, [1035].log_data[0].max := 1.0, [1035].log_data[0].total := 300.0, [1035].log_data[0].time := 300.0, [1035].log_data[0].minminute := 35, [1035].log_data[0].maxminute := 35, [1035].log_data[0].valid := 1, [1035].log_data[1].valid := 1, [1035].log_data[2].valid := 1, [1035].log_data[3].valid := 1, [1035].log_data[4].valid := 1, [1035].log_data[5].valid := 1, [1035].log_data[6].valid := 1, [1035].log_data[7].valid := 1, [1035].log_data[8].valid := 1, [1035].log_data[9].valid := 1, [1035].log_data[10].valid := 1, [1035].log_data[11].valid := 1, [1035].log_data[12].valid := 1, [1035].log_data[13].valid := 1, [1035].log_data[14].valid := 1, [1035].log_data[15].valid := 1, [1035].log_data[16].valid := 1, [1035].log_data[17].valid := 1, [1035].log_data[18].valid := 1, [1035].log_data[19].valid := 1, [1035].time.Year := 2023, [1035].time.Month := 1, [1035].time.Day := 13, [1035].time.Hour := 6, [1035].time.Minute := 39, [1035].time.Second := 59, [1036].log_data[0].min := 1.0, [1036].log_data[0].max := 1.0, [1036].log_data[0].total := 300.0, [1036].log_data[0].time := 300.0, [1036].log_data[0].minminute := 40, [1036].log_data[0].maxminute := 40, [1036].log_data[0].valid := 1, [1036].log_data[1].valid := 1, [1036].log_data[2].valid := 1, [1036].log_data[3].valid := 1,
        [1036].log_data[4].valid := 1, [1036].log_data[5].valid := 1, [1036].log_data[6].valid := 1, [1036].log_data[7].valid := 1, [1036].log_data[8].valid := 1, [1036].log_data[9].valid := 1, [1036].log_data[10].valid := 1, [1036].log_data[11].valid := 1, [1036].log_data[12].valid := 1, [1036].log_data[13].valid := 1, [1036].log_data[14].valid := 1, [1036].log_data[15].valid := 1, [1036].log_data[16].valid := 1, [1036].log_data[17].valid := 1, [1036].log_data[18].valid := 1, [1036].log_data[19].valid := 1, [1036].time.Year := 2023, [1036].time.Month := 1, [1036].time.Day := 13, [1036].time.Hour := 6, [1036].time.Minute := 44, [1036].time.Second := 59, [1037].log_data[0].min := 1.0, [1037].log_data[0].max := 1.0, [1037].log_data[0].total := 300.0, [1037].log_data[0].time := 300.0, [1037].log_data[0].minminute := 45, [1037].log_data[0].maxminute := 45, [1037].log_data[0].valid := 1, [1037].log_data[1].valid := 1, [1037].log_data[2].valid := 1, [1037].log_data[3].valid := 1, [1037].log_data[4].valid := 1, [1037].log_data[5].valid := 1, [1037].log_data[6].valid := 1, [1037].log_data[7].valid := 1, [1037].log_data[8].valid := 1, [1037].log_data[9].valid := 1, [1037].log_data[10].valid := 1, [1037].log_data[11].valid := 1, [1037].log_data[12].valid := 1, [1037].log_data[13].valid := 1, [1037].log_data[14].valid := 1, [1037].log_data[15].valid := 1, [1037].log_data[16].valid := 1, [1037].log_data[17].valid := 1, [1037].log_data[18].valid := 1, [1037].log_data[19].valid := 1, [1037].time.Year := 2023, [1037].time.Month := 1, [1037].time.Day := 13, [1037].time.Hour := 6, [1037].time.Minute := 49, [1037].time.Second := 59, [1038].log_data[0].min := 1.0, [1038].log_data[0].max := 1.0, [1038].log_data[0].total := 300.0, [1038].log_data[0].time := 300.0, [1038].log_data[0].minminute := 50, [1038].log_data[0].maxminute := 50,
        [1038].log_data[0].valid := 1, [1038].log_data[1].valid := 1, [1038].log_data[2].valid := 1, [1038].log_data[3].valid := 1, [1038].log_data[4].valid := 1, [1038].log_data[5].valid := 1, [1038].log_data[6].valid := 1, [1038].log_data[7].valid := 1, [1038].log_data[8].valid := 1, [1038].log_data[9].valid := 1, [1038].log_data[10].valid := 1, [1038].log_data[11].valid := 1, [1038].log_data[12].valid := 1, [1038].log_data[13].valid := 1, [1038].log_data[14].valid := 1, [1038].log_data[15].valid := 1, [1038].log_data[16].valid := 1, [1038].log_data[17].valid := 1, [1038].log_data[18].valid := 1, [1038].log_data[19].valid := 1, [1038].time.Year := 2023, [1038].time.Month := 1, [1038].time.Day := 13, [1038].time.Hour := 6, [1038].time.Minute := 54, [1038].time.Second := 59, [1039].log_data[0].min := 1.0, [1039].log_data[0].max := 1.0, [1039].log_data[0].total := 300.0, [1039].log_data[0].time := 300.0, [1039].log_data[0].minminute := 55, [1039].log_data[0].maxminute := 55, [1039].log_data[0].valid := 1, [1039].log_data[1].valid := 1, [1039].log_data[2].valid := 1, [1039].log_data[3].valid := 1, [1039].log_data[4].valid := 1, [1039].log_data[5].valid := 1, [1039].log_data[6].valid := 1, [1039].log_data[7].valid := 1, [1039].log_data[8].valid := 1, [1039].log_data[9].valid := 1, [1039].log_data[10].valid := 1, [1039].log_data[11].valid := 1, [1039].log_data[12].valid := 1, [1039].log_data[13].valid := 1, [1039].log_data[14].valid := 1, [1039].log_data[15].valid := 1, [1039].log_data[16].valid := 1, [1039].log_data[17].valid := 1, [1039].log_data[18].valid := 1, [1039].log_data[19].valid := 1, [1039].time.Year := 2023, [1039].time.Month := 1, [1039].time.Day := 13, [1039].time.Hour := 6, [1039].time.Minute := 59, [1039].time.Second := 59, [1040].log_data[0].min := 1.0, [1040].log_data[0].max := 1.0,
        [1040].log_data[0].total := 300.0, [1040].log_data[0].time := 300.0, [1040].log_data[0].valid := 1, [1040].log_data[1].valid := 1, [1040].log_data[2].valid := 1, [1040].log_data[3].valid := 1, [1040].log_data[4].valid := 1, [1040].log_data[5].valid := 1, [1040].log_data[6].valid := 1, [1040].log_data[7].valid := 1, [1040].log_data[8].valid := 1, [1040].log_data[9].valid := 1, [1040].log_data[10].valid := 1, [1040].log_data[11].valid := 1, [1040].log_data[12].valid := 1, [1040].log_data[13].valid := 1, [1040].log_data[14].valid := 1, [1040].log_data[15].valid := 1, [1040].log_data[16].valid := 1, [1040].log_data[17].valid := 1, [1040].log_data[18].valid := 1, [1040].log_data[19].valid := 1, [1040].time.Year := 2023, [1040].time.Month := 1, [1040].time.Day := 13, [1040].time.Hour := 7, [1040].time.Minute := 4, [1040].time.Second := 59, [1041].log_data[0].min := 1.0, [1041].log_data[0].max := 1.0, [1041].log_data[0].total := 300.0, [1041].log_data[0].time := 300.0, [1041].log_data[0].minminute := 5, [1041].log_data[0].maxminute := 5, [1041].log_data[0].valid := 1, [1041].log_data[1].valid := 1, [1041].log_data[2].valid := 1, [1041].log_data[3].valid := 1, [1041].log_data[4].valid := 1, [1041].log_data[5].valid := 1, [1041].log_data[6].valid := 1, [1041].log_data[7].valid := 1, [1041].log_data[8].valid := 1, [1041].log_data[9].valid := 1, [1041].log_data[10].valid := 1, [1041].log_data[11].valid := 1, [1041].log_data[12].valid := 1, [1041].log_data[13].valid := 1, [1041].log_data[14].valid := 1, [1041].log_data[15].valid := 1, [1041].log_data[16].valid := 1, [1041].log_data[17].valid := 1, [1041].log_data[18].valid := 1, [1041].log_data[19].valid := 1, [1041].time.Year := 2023, [1041].time.Month := 1, [1041].time.Day := 13, [1041].time.Hour := 7, [1041].time.Minute := 9, [1041].time.Second := 59,
        [1042].log_data[0].min := 1.0, [1042].log_data[0].max := 1.0, [1042].log_data[0].total := 300.0, [1042].log_data[0].time := 300.0, [1042].log_data[0].minminute := 10, [1042].log_data[0].maxminute := 10, [1042].log_data[0].valid := 1, [1042].log_data[1].valid := 1, [1042].log_data[2].valid := 1, [1042].log_data[3].valid := 1, [1042].log_data[4].valid := 1, [1042].log_data[5].valid := 1, [1042].log_data[6].valid := 1, [1042].log_data[7].valid := 1, [1042].log_data[8].valid := 1, [1042].log_data[9].valid := 1, [1042].log_data[10].valid := 1, [1042].log_data[11].valid := 1, [1042].log_data[12].valid := 1, [1042].log_data[13].valid := 1, [1042].log_data[14].valid := 1, [1042].log_data[15].valid := 1, [1042].log_data[16].valid := 1, [1042].log_data[17].valid := 1, [1042].log_data[18].valid := 1, [1042].log_data[19].valid := 1, [1042].time.Year := 2023, [1042].time.Month := 1, [1042].time.Day := 13, [1042].time.Hour := 7, [1042].time.Minute := 14, [1042].time.Second := 59, [1043].log_data[0].min := 1.0, [1043].log_data[0].max := 1.0, [1043].log_data[0].total := 300.0, [1043].log_data[0].time := 300.0, [1043].log_data[0].minminute := 15, [1043].log_data[0].maxminute := 15, [1043].log_data[0].valid := 1, [1043].log_data[1].valid := 1, [1043].log_data[2].valid := 1, [1043].log_data[3].valid := 1, [1043].log_data[4].valid := 1, [1043].log_data[5].valid := 1, [1043].log_data[6].valid := 1, [1043].log_data[7].valid := 1, [1043].log_data[8].valid := 1, [1043].log_data[9].valid := 1, [1043].log_data[10].valid := 1, [1043].log_data[11].valid := 1, [1043].log_data[12].valid := 1, [1043].log_data[13].valid := 1, [1043].log_data[14].valid := 1, [1043].log_data[15].valid := 1, [1043].log_data[16].valid := 1, [1043].log_data[17].valid := 1, [1043].log_data[18].valid := 1, [1043].log_data[19].valid := 1, [1043].time.Year := 2023, [1043].time.Month := 1,
        [1043].time.Day := 13, [1043].time.Hour := 7, [1043].time.Minute := 19, [1043].time.Second := 59, [1044].log_data[0].min := 1.0, [1044].log_data[0].max := 1.0, [1044].log_data[0].total := 300.0, [1044].log_data[0].time := 300.0, [1044].log_data[0].minminute := 20, [1044].log_data[0].maxminute := 20, [1044].log_data[0].valid := 1, [1044].log_data[1].valid := 1, [1044].log_data[2].valid := 1, [1044].log_data[3].valid := 1, [1044].log_data[4].valid := 1, [1044].log_data[5].valid := 1, [1044].log_data[6].valid := 1, [1044].log_data[7].valid := 1, [1044].log_data[8].valid := 1, [1044].log_data[9].valid := 1, [1044].log_data[10].valid := 1, [1044].log_data[11].valid := 1, [1044].log_data[12].valid := 1, [1044].log_data[13].valid := 1, [1044].log_data[14].valid := 1, [1044].log_data[15].valid := 1, [1044].log_data[16].valid := 1, [1044].log_data[17].valid := 1, [1044].log_data[18].valid := 1, [1044].log_data[19].valid := 1, [1044].time.Year := 2023, [1044].time.Month := 1, [1044].time.Day := 13, [1044].time.Hour := 7, [1044].time.Minute := 24, [1044].time.Second := 59, [1045].log_data[0].min := 1.0, [1045].log_data[0].max := 1.0, [1045].log_data[0].total := 300.0, [1045].log_data[0].time := 300.0, [1045].log_data[0].minminute := 25, [1045].log_data[0].maxminute := 25, [1045].log_data[0].valid := 1, [1045].log_data[1].valid := 1, [1045].log_data[2].valid := 1, [1045].log_data[3].valid := 1, [1045].log_data[4].valid := 1, [1045].log_data[5].valid := 1, [1045].log_data[6].valid := 1, [1045].log_data[7].valid := 1, [1045].log_data[8].valid := 1, [1045].log_data[9].valid := 1, [1045].log_data[10].valid := 1, [1045].log_data[11].valid := 1, [1045].log_data[12].valid := 1, [1045].log_data[13].valid := 1, [1045].log_data[14].valid := 1, [1045].log_data[15].valid := 1, [1045].log_data[16].valid := 1, [1045].log_data[17].valid := 1,
        [1045].log_data[18].valid := 1, [1045].log_data[19].valid := 1, [1045].time.Year := 2023, [1045].time.Month := 1, [1045].time.Day := 13, [1045].time.Hour := 7, [1045].time.Minute := 29, [1045].time.Second := 59, [1046].log_data[0].min := 1.0, [1046].log_data[0].max := 1.0, [1046].log_data[0].total := 300.0, [1046].log_data[0].time := 300.0, [1046].log_data[0].minminute := 30, [1046].log_data[0].maxminute := 30, [1046].log_data[0].valid := 1, [1046].log_data[1].valid := 1, [1046].log_data[2].valid := 1, [1046].log_data[3].valid := 1, [1046].log_data[4].valid := 1, [1046].log_data[5].valid := 1, [1046].log_data[6].valid := 1, [1046].log_data[7].valid := 1, [1046].log_data[8].valid := 1, [1046].log_data[9].valid := 1, [1046].log_data[10].valid := 1, [1046].log_data[11].valid := 1, [1046].log_data[12].valid := 1, [1046].log_data[13].valid := 1, [1046].log_data[14].valid := 1, [1046].log_data[15].valid := 1, [1046].log_data[16].valid := 1, [1046].log_data[17].valid := 1, [1046].log_data[18].valid := 1, [1046].log_data[19].valid := 1, [1046].time.Year := 2023, [1046].time.Month := 1, [1046].time.Day := 13, [1046].time.Hour := 7, [1046].time.Minute := 34, [1046].time.Second := 59, [1047].log_data[0].min := 1.0, [1047].log_data[0].max := 1.0, [1047].log_data[0].total := 300.0, [1047].log_data[0].time := 300.0, [1047].log_data[0].minminute := 35, [1047].log_data[0].maxminute := 35, [1047].log_data[0].valid := 1, [1047].log_data[1].valid := 1, [1047].log_data[2].valid := 1, [1047].log_data[3].valid := 1, [1047].log_data[4].valid := 1, [1047].log_data[5].valid := 1, [1047].log_data[6].valid := 1, [1047].log_data[7].valid := 1, [1047].log_data[8].valid := 1, [1047].log_data[9].valid := 1, [1047].log_data[10].valid := 1, [1047].log_data[11].valid := 1, [1047].log_data[12].valid := 1, [1047].log_data[13].valid := 1,
        [1047].log_data[14].valid := 1, [1047].log_data[15].valid := 1, [1047].log_data[16].valid := 1, [1047].log_data[17].valid := 1, [1047].log_data[18].valid := 1, [1047].log_data[19].valid := 1, [1047].time.Year := 2023, [1047].time.Month := 1, [1047].time.Day := 13, [1047].time.Hour := 7, [1047].time.Minute := 39, [1047].time.Second := 59, [1048].log_data[0].min := 1.0, [1048].log_data[0].max := 1.0, [1048].log_data[0].total := 300.0, [1048].log_data[0].time := 300.0, [1048].log_data[0].minminute := 40, [1048].log_data[0].maxminute := 40, [1048].log_data[0].valid := 1, [1048].log_data[1].valid := 1, [1048].log_data[2].valid := 1, [1048].log_data[3].valid := 1, [1048].log_data[4].valid := 1, [1048].log_data[5].valid := 1, [1048].log_data[6].valid := 1, [1048].log_data[7].valid := 1, [1048].log_data[8].valid := 1, [1048].log_data[9].valid := 1, [1048].log_data[10].valid := 1, [1048].log_data[11].valid := 1, [1048].log_data[12].valid := 1, [1048].log_data[13].valid := 1, [1048].log_data[14].valid := 1, [1048].log_data[15].valid := 1, [1048].log_data[16].valid := 1, [1048].log_data[17].valid := 1, [1048].log_data[18].valid := 1, [1048].log_data[19].valid := 1, [1048].time.Year := 2023, [1048].time.Month := 1, [1048].time.Day := 13, [1048].time.Hour := 7, [1048].time.Minute := 44, [1048].time.Second := 59, [1049].log_data[0].min := 1.0, [1049].log_data[0].max := 1.0, [1049].log_data[0].total := 300.0, [1049].log_data[0].time := 300.0, [1049].log_data[0].minminute := 45, [1049].log_data[0].maxminute := 45, [1049].log_data[0].valid := 1, [1049].log_data[1].valid := 1, [1049].log_data[2].valid := 1, [1049].log_data[3].valid := 1, [1049].log_data[4].valid := 1, [1049].log_data[5].valid := 1, [1049].log_data[6].valid := 1, [1049].log_data[7].valid := 1, [1049].log_data[8].valid := 1, [1049].log_data[9].valid := 1,
        [1049].log_data[10].valid := 1, [1049].log_data[11].valid := 1, [1049].log_data[12].valid := 1, [1049].log_data[13].valid := 1, [1049].log_data[14].valid := 1, [1049].log_data[15].valid := 1, [1049].log_data[16].valid := 1, [1049].log_data[17].valid := 1, [1049].log_data[18].valid := 1, [1049].log_data[19].valid := 1, [1049].time.Year := 2023, [1049].time.Month := 1, [1049].time.Day := 13, [1049].time.Hour := 7, [1049].time.Minute := 49, [1049].time.Second := 59, [1050].log_data[0].min := 1.0, [1050].log_data[0].max := 1.0, [1050].log_data[0].total := 300.0, [1050].log_data[0].time := 300.0, [1050].log_data[0].minminute := 50, [1050].log_data[0].maxminute := 50, [1050].log_data[0].valid := 1, [1050].log_data[1].valid := 1, [1050].log_data[2].valid := 1, [1050].log_data[3].valid := 1, [1050].log_data[4].valid := 1, [1050].log_data[5].valid := 1, [1050].log_data[6].valid := 1, [1050].log_data[7].valid := 1, [1050].log_data[8].valid := 1, [1050].log_data[9].valid := 1, [1050].log_data[10].valid := 1, [1050].log_data[11].valid := 1, [1050].log_data[12].valid := 1, [1050].log_data[13].valid := 1, [1050].log_data[14].valid := 1, [1050].log_data[15].valid := 1, [1050].log_data[16].valid := 1, [1050].log_data[17].valid := 1, [1050].log_data[18].valid := 1, [1050].log_data[19].valid := 1, [1050].time.Year := 2023, [1050].time.Month := 1, [1050].time.Day := 13, [1050].time.Hour := 7, [1050].time.Minute := 54, [1050].time.Second := 59, [1051].log_data[0].min := 1.0, [1051].log_data[0].max := 1.0, [1051].log_data[0].total := 300.0, [1051].log_data[0].time := 300.0, [1051].log_data[0].minminute := 55, [1051].log_data[0].maxminute := 55, [1051].log_data[0].valid := 1, [1051].log_data[1].valid := 1, [1051].log_data[2].valid := 1, [1051].log_data[3].valid := 1, [1051].log_data[4].valid := 1, [1051].log_data[5].valid := 1,
        [1051].log_data[6].valid := 1, [1051].log_data[7].valid := 1, [1051].log_data[8].valid := 1, [1051].log_data[9].valid := 1, [1051].log_data[10].valid := 1, [1051].log_data[11].valid := 1, [1051].log_data[12].valid := 1, [1051].log_data[13].valid := 1, [1051].log_data[14].valid := 1, [1051].log_data[15].valid := 1, [1051].log_data[16].valid := 1, [1051].log_data[17].valid := 1, [1051].log_data[18].valid := 1, [1051].log_data[19].valid := 1, [1051].time.Year := 2023, [1051].time.Month := 1, [1051].time.Day := 13, [1051].time.Hour := 7, [1051].time.Minute := 59, [1051].time.Second := 59, [1052].log_data[0].min := 1.0, [1052].log_data[0].max := 1.0, [1052].log_data[0].total := 300.0, [1052].log_data[0].time := 300.0, [1052].log_data[0].valid := 1, [1052].log_data[1].valid := 1, [1052].log_data[2].valid := 1, [1052].log_data[3].valid := 1, [1052].log_data[4].valid := 1, [1052].log_data[5].valid := 1, [1052].log_data[6].valid := 1, [1052].log_data[7].valid := 1, [1052].log_data[8].valid := 1, [1052].log_data[9].valid := 1, [1052].log_data[10].valid := 1, [1052].log_data[11].valid := 1, [1052].log_data[12].valid := 1, [1052].log_data[13].valid := 1, [1052].log_data[14].valid := 1, [1052].log_data[15].valid := 1, [1052].log_data[16].valid := 1, [1052].log_data[17].valid := 1, [1052].log_data[18].valid := 1, [1052].log_data[19].valid := 1, [1052].time.Year := 2023, [1052].time.Month := 1, [1052].time.Day := 13, [1052].time.Hour := 8, [1052].time.Minute := 4, [1052].time.Second := 59, [1053].log_data[0].min := 1.0, [1053].log_data[0].max := 1.0, [1053].log_data[0].total := 300.0, [1053].log_data[0].time := 300.0, [1053].log_data[0].minminute := 5, [1053].log_data[0].maxminute := 5, [1053].log_data[0].valid := 1, [1053].log_data[1].valid := 1, [1053].log_data[2].valid := 1, [1053].log_data[3].valid := 1,
        [1053].log_data[4].valid := 1, [1053].log_data[5].valid := 1, [1053].log_data[6].valid := 1, [1053].log_data[7].valid := 1, [1053].log_data[8].valid := 1, [1053].log_data[9].valid := 1, [1053].log_data[10].valid := 1, [1053].log_data[11].valid := 1, [1053].log_data[12].valid := 1, [1053].log_data[13].valid := 1, [1053].log_data[14].valid := 1, [1053].log_data[15].valid := 1, [1053].log_data[16].valid := 1, [1053].log_data[17].valid := 1, [1053].log_data[18].valid := 1, [1053].log_data[19].valid := 1, [1053].time.Year := 2023, [1053].time.Month := 1, [1053].time.Day := 13, [1053].time.Hour := 8, [1053].time.Minute := 9, [1053].time.Second := 59, [1054].log_data[0].min := 1.0, [1054].log_data[0].max := 1.0, [1054].log_data[0].total := 300.0, [1054].log_data[0].time := 300.0, [1054].log_data[0].minminute := 10, [1054].log_data[0].maxminute := 10, [1054].log_data[0].valid := 1, [1054].log_data[1].valid := 1, [1054].log_data[2].valid := 1, [1054].log_data[3].valid := 1, [1054].log_data[4].valid := 1, [1054].log_data[5].valid := 1, [1054].log_data[6].valid := 1, [1054].log_data[7].valid := 1, [1054].log_data[8].valid := 1, [1054].log_data[9].valid := 1, [1054].log_data[10].valid := 1, [1054].log_data[11].valid := 1, [1054].log_data[12].valid := 1, [1054].log_data[13].valid := 1, [1054].log_data[14].valid := 1, [1054].log_data[15].valid := 1, [1054].log_data[16].valid := 1, [1054].log_data[17].valid := 1, [1054].log_data[18].valid := 1, [1054].log_data[19].valid := 1, [1054].time.Year := 2023, [1054].time.Month := 1, [1054].time.Day := 13, [1054].time.Hour := 8, [1054].time.Minute := 14, [1054].time.Second := 59, [1055].log_data[0].min := 1.0, [1055].log_data[0].max := 1.0, [1055].log_data[0].total := 300.0, [1055].log_data[0].time := 300.0, [1055].log_data[0].minminute := 15, [1055].log_data[0].maxminute := 15,
        [1055].log_data[0].valid := 1, [1055].log_data[1].valid := 1, [1055].log_data[2].valid := 1, [1055].log_data[3].valid := 1, [1055].log_data[4].valid := 1, [1055].log_data[5].valid := 1, [1055].log_data[6].valid := 1, [1055].log_data[7].valid := 1, [1055].log_data[8].valid := 1, [1055].log_data[9].valid := 1, [1055].log_data[10].valid := 1, [1055].log_data[11].valid := 1, [1055].log_data[12].valid := 1, [1055].log_data[13].valid := 1, [1055].log_data[14].valid := 1, [1055].log_data[15].valid := 1, [1055].log_data[16].valid := 1, [1055].log_data[17].valid := 1, [1055].log_data[18].valid := 1, [1055].log_data[19].valid := 1, [1055].time.Year := 2023, [1055].time.Month := 1, [1055].time.Day := 13, [1055].time.Hour := 8, [1055].time.Minute := 19, [1055].time.Second := 59, [1056].log_data[0].min := 1.0, [1056].log_data[0].max := 1.0, [1056].log_data[0].total := 300.0, [1056].log_data[0].time := 300.0, [1056].log_data[0].minminute := 20, [1056].log_data[0].maxminute := 20, [1056].log_data[0].valid := 1, [1056].log_data[1].valid := 1, [1056].log_data[2].valid := 1, [1056].log_data[3].valid := 1, [1056].log_data[4].valid := 1, [1056].log_data[5].valid := 1, [1056].log_data[6].valid := 1, [1056].log_data[7].valid := 1, [1056].log_data[8].valid := 1, [1056].log_data[9].valid := 1, [1056].log_data[10].valid := 1, [1056].log_data[11].valid := 1, [1056].log_data[12].valid := 1, [1056].log_data[13].valid := 1, [1056].log_data[14].valid := 1, [1056].log_data[15].valid := 1, [1056].log_data[16].valid := 1, [1056].log_data[17].valid := 1, [1056].log_data[18].valid := 1, [1056].log_data[19].valid := 1, [1056].time.Year := 2023, [1056].time.Month := 1, [1056].time.Day := 13, [1056].time.Hour := 8, [1056].time.Minute := 24, [1056].time.Second := 59, [1057].log_data[0].min := 1.0, [1057].log_data[0].max := 1.0,
        [1057].log_data[0].total := 300.0, [1057].log_data[0].time := 300.0, [1057].log_data[0].minminute := 25, [1057].log_data[0].maxminute := 25, [1057].log_data[0].valid := 1, [1057].log_data[1].valid := 1, [1057].log_data[2].valid := 1, [1057].log_data[3].valid := 1, [1057].log_data[4].valid := 1, [1057].log_data[5].valid := 1, [1057].log_data[6].valid := 1, [1057].log_data[7].valid := 1, [1057].log_data[8].valid := 1, [1057].log_data[9].valid := 1, [1057].log_data[10].valid := 1, [1057].log_data[11].valid := 1, [1057].log_data[12].valid := 1, [1057].log_data[13].valid := 1, [1057].log_data[14].valid := 1, [1057].log_data[15].valid := 1, [1057].log_data[16].valid := 1, [1057].log_data[17].valid := 1, [1057].log_data[18].valid := 1, [1057].log_data[19].valid := 1, [1057].time.Year := 2023, [1057].time.Month := 1, [1057].time.Day := 13, [1057].time.Hour := 8, [1057].time.Minute := 29, [1057].time.Second := 59, [1058].log_data[0].min := 1.0, [1058].log_data[0].max := 1.0, [1058].log_data[0].total := 300.0, [1058].log_data[0].time := 300.0, [1058].log_data[0].minminute := 30, [1058].log_data[0].maxminute := 30, [1058].log_data[0].valid := 1, [1058].log_data[1].valid := 1, [1058].log_data[2].valid := 1, [1058].log_data[3].valid := 1, [1058].log_data[4].valid := 1, [1058].log_data[5].valid := 1, [1058].log_data[6].valid := 1, [1058].log_data[7].valid := 1, [1058].log_data[8].valid := 1, [1058].log_data[9].valid := 1, [1058].log_data[10].valid := 1, [1058].log_data[11].valid := 1, [1058].log_data[12].valid := 1, [1058].log_data[13].valid := 1, [1058].log_data[14].valid := 1, [1058].log_data[15].valid := 1, [1058].log_data[16].valid := 1, [1058].log_data[17].valid := 1, [1058].log_data[18].valid := 1, [1058].log_data[19].valid := 1, [1058].time.Year := 2023, [1058].time.Month := 1, [1058].time.Day := 13, [1058].time.Hour := 8,
        [1058].time.Minute := 34, [1058].time.Second := 59, [1059].log_data[0].min := 1.0, [1059].log_data[0].max := 1.0, [1059].log_data[0].total := 300.0, [1059].log_data[0].time := 300.0, [1059].log_data[0].minminute := 35, [1059].log_data[0].maxminute := 35, [1059].log_data[0].valid := 1, [1059].log_data[1].valid := 1, [1059].log_data[2].valid := 1, [1059].log_data[3].valid := 1, [1059].log_data[4].valid := 1, [1059].log_data[5].valid := 1, [1059].log_data[6].valid := 1, [1059].log_data[7].valid := 1, [1059].log_data[8].valid := 1, [1059].log_data[9].valid := 1, [1059].log_data[10].valid := 1, [1059].log_data[11].valid := 1, [1059].log_data[12].valid := 1, [1059].log_data[13].valid := 1, [1059].log_data[14].valid := 1, [1059].log_data[15].valid := 1, [1059].log_data[16].valid := 1, [1059].log_data[17].valid := 1, [1059].log_data[18].valid := 1, [1059].log_data[19].valid := 1, [1059].time.Year := 2023, [1059].time.Month := 1, [1059].time.Day := 13, [1059].time.Hour := 8, [1059].time.Minute := 39, [1059].time.Second := 59, [1060].log_data[0].min := 1.0, [1060].log_data[0].max := 1.0, [1060].log_data[0].total := 300.0, [1060].log_data[0].time := 300.0, [1060].log_data[0].minminute := 40, [1060].log_data[0].maxminute := 40, [1060].log_data[0].valid := 1, [1060].log_data[1].valid := 1, [1060].log_data[2].valid := 1, [1060].log_data[3].valid := 1, [1060].log_data[4].valid := 1, [1060].log_data[5].valid := 1, [1060].log_data[6].valid := 1, [1060].log_data[7].valid := 1, [1060].log_data[8].valid := 1, [1060].log_data[9].valid := 1, [1060].log_data[10].valid := 1, [1060].log_data[11].valid := 1, [1060].log_data[12].valid := 1, [1060].log_data[13].valid := 1, [1060].log_data[14].valid := 1, [1060].log_data[15].valid := 1, [1060].log_data[16].valid := 1, [1060].log_data[17].valid := 1, [1060].log_data[18].valid := 1, [1060].log_data[19].valid := 1,
        [1060].time.Year := 2023, [1060].time.Month := 1, [1060].time.Day := 13, [1060].time.Hour := 8, [1060].time.Minute := 44, [1060].time.Second := 59, [1061].log_data[0].min := 1.0, [1061].log_data[0].max := 1.0, [1061].log_data[0].total := 300.0, [1061].log_data[0].time := 300.0, [1061].log_data[0].minminute := 45, [1061].log_data[0].maxminute := 45, [1061].log_data[0].valid := 1, [1061].log_data[1].valid := 1, [1061].log_data[2].valid := 1, [1061].log_data[3].valid := 1, [1061].log_data[4].valid := 1, [1061].log_data[5].valid := 1, [1061].log_data[6].valid := 1, [1061].log_data[7].valid := 1, [1061].log_data[8].valid := 1, [1061].log_data[9].valid := 1, [1061].log_data[10].valid := 1, [1061].log_data[11].valid := 1, [1061].log_data[12].valid := 1, [1061].log_data[13].valid := 1, [1061].log_data[14].valid := 1, [1061].log_data[15].valid := 1, [1061].log_data[16].valid := 1, [1061].log_data[17].valid := 1, [1061].log_data[18].valid := 1, [1061].log_data[19].valid := 1, [1061].time.Year := 2023, [1061].time.Month := 1, [1061].time.Day := 13, [1061].time.Hour := 8, [1061].time.Minute := 49, [1061].time.Second := 59, [1062].log_data[0].min := 1.0, [1062].log_data[0].max := 1.0, [1062].log_data[0].total := 300.0, [1062].log_data[0].time := 300.0, [1062].log_data[0].minminute := 50, [1062].log_data[0].maxminute := 50, [1062].log_data[0].valid := 1, [1062].log_data[1].valid := 1, [1062].log_data[2].valid := 1, [1062].log_data[3].valid := 1, [1062].log_data[4].valid := 1, [1062].log_data[5].valid := 1, [1062].log_data[6].valid := 1, [1062].log_data[7].valid := 1, [1062].log_data[8].valid := 1, [1062].log_data[9].valid := 1, [1062].log_data[10].valid := 1, [1062].log_data[11].valid := 1, [1062].log_data[12].valid := 1, [1062].log_data[13].valid := 1, [1062].log_data[14].valid := 1, [1062].log_data[15].valid := 1,
        [1062].log_data[16].valid := 1, [1062].log_data[17].valid := 1, [1062].log_data[18].valid := 1, [1062].log_data[19].valid := 1, [1062].time.Year := 2023, [1062].time.Month := 1, [1062].time.Day := 13, [1062].time.Hour := 8, [1062].time.Minute := 54, [1062].time.Second := 59, [1063].log_data[0].min := 1.0, [1063].log_data[0].max := 1.0, [1063].log_data[0].total := 300.0, [1063].log_data[0].time := 300.0, [1063].log_data[0].minminute := 55, [1063].log_data[0].maxminute := 55, [1063].log_data[0].valid := 1, [1063].log_data[1].valid := 1, [1063].log_data[2].valid := 1, [1063].log_data[3].valid := 1, [1063].log_data[4].valid := 1, [1063].log_data[5].valid := 1, [1063].log_data[6].valid := 1, [1063].log_data[7].valid := 1, [1063].log_data[8].valid := 1, [1063].log_data[9].valid := 1, [1063].log_data[10].valid := 1, [1063].log_data[11].valid := 1, [1063].log_data[12].valid := 1, [1063].log_data[13].valid := 1, [1063].log_data[14].valid := 1, [1063].log_data[15].valid := 1, [1063].log_data[16].valid := 1, [1063].log_data[17].valid := 1, [1063].log_data[18].valid := 1, [1063].log_data[19].valid := 1, [1063].time.Year := 2023, [1063].time.Month := 1, [1063].time.Day := 13, [1063].time.Hour := 8, [1063].time.Minute := 59, [1063].time.Second := 59, [1064].log_data[0].min := 1.0, [1064].log_data[0].max := 1.0, [1064].log_data[0].total := 300.0, [1064].log_data[0].time := 300.0, [1064].log_data[0].valid := 1, [1064].log_data[1].valid := 1, [1064].log_data[2].valid := 1, [1064].log_data[3].valid := 1, [1064].log_data[4].valid := 1, [1064].log_data[5].valid := 1, [1064].log_data[6].valid := 1, [1064].log_data[7].valid := 1, [1064].log_data[8].valid := 1, [1064].log_data[9].valid := 1, [1064].log_data[10].valid := 1, [1064].log_data[11].valid := 1, [1064].log_data[12].valid := 1, [1064].log_data[13].valid := 1,
        [1064].log_data[14].valid := 1, [1064].log_data[15].valid := 1, [1064].log_data[16].valid := 1, [1064].log_data[17].valid := 1, [1064].log_data[18].valid := 1, [1064].log_data[19].valid := 1, [1064].time.Year := 2023, [1064].time.Month := 1, [1064].time.Day := 13, [1064].time.Hour := 9, [1064].time.Minute := 4, [1064].time.Second := 59, [1065].log_data[0].min := 1.0, [1065].log_data[0].max := 1.0, [1065].log_data[0].total := 300.0, [1065].log_data[0].time := 300.0, [1065].log_data[0].minminute := 5, [1065].log_data[0].maxminute := 5, [1065].log_data[0].valid := 1, [1065].log_data[1].valid := 1, [1065].log_data[2].valid := 1, [1065].log_data[3].valid := 1, [1065].log_data[4].valid := 1, [1065].log_data[5].valid := 1, [1065].log_data[6].valid := 1, [1065].log_data[7].valid := 1, [1065].log_data[8].valid := 1, [1065].log_data[9].valid := 1, [1065].log_data[10].valid := 1, [1065].log_data[11].valid := 1, [1065].log_data[12].valid := 1, [1065].log_data[13].valid := 1, [1065].log_data[14].valid := 1, [1065].log_data[15].valid := 1, [1065].log_data[16].valid := 1, [1065].log_data[17].valid := 1, [1065].log_data[18].valid := 1, [1065].log_data[19].valid := 1, [1065].time.Year := 2023, [1065].time.Month := 1, [1065].time.Day := 13, [1065].time.Hour := 9, [1065].time.Minute := 9, [1065].time.Second := 59, [1066].log_data[0].min := 1.0, [1066].log_data[0].max := 1.0, [1066].log_data[0].total := 300.0, [1066].log_data[0].time := 300.0, [1066].log_data[0].minminute := 10, [1066].log_data[0].maxminute := 10, [1066].log_data[0].valid := 1, [1066].log_data[1].valid := 1, [1066].log_data[2].valid := 1, [1066].log_data[3].valid := 1, [1066].log_data[4].valid := 1, [1066].log_data[5].valid := 1, [1066].log_data[6].valid := 1, [1066].log_data[7].valid := 1, [1066].log_data[8].valid := 1, [1066].log_data[9].valid := 1,
        [1066].log_data[10].valid := 1, [1066].log_data[11].valid := 1, [1066].log_data[12].valid := 1, [1066].log_data[13].valid := 1, [1066].log_data[14].valid := 1, [1066].log_data[15].valid := 1, [1066].log_data[16].valid := 1, [1066].log_data[17].valid := 1, [1066].log_data[18].valid := 1, [1066].log_data[19].valid := 1, [1066].time.Year := 2023, [1066].time.Month := 1, [1066].time.Day := 13, [1066].time.Hour := 9, [1066].time.Minute := 14, [1066].time.Second := 59, [1067].log_data[0].min := 1.0, [1067].log_data[0].max := 1.0, [1067].log_data[0].total := 300.0, [1067].log_data[0].time := 300.0, [1067].log_data[0].minminute := 15, [1067].log_data[0].maxminute := 15, [1067].log_data[0].valid := 1, [1067].log_data[1].valid := 1, [1067].log_data[2].valid := 1, [1067].log_data[3].valid := 1, [1067].log_data[4].valid := 1, [1067].log_data[5].valid := 1, [1067].log_data[6].valid := 1, [1067].log_data[7].valid := 1, [1067].log_data[8].valid := 1, [1067].log_data[9].valid := 1, [1067].log_data[10].valid := 1, [1067].log_data[11].valid := 1, [1067].log_data[12].valid := 1, [1067].log_data[13].valid := 1, [1067].log_data[14].valid := 1, [1067].log_data[15].valid := 1, [1067].log_data[16].valid := 1, [1067].log_data[17].valid := 1, [1067].log_data[18].valid := 1, [1067].log_data[19].valid := 1, [1067].time.Year := 2023, [1067].time.Month := 1, [1067].time.Day := 13, [1067].time.Hour := 9, [1067].time.Minute := 19, [1067].time.Second := 59, [1068].log_data[0].min := 1.0, [1068].log_data[0].max := 1.0, [1068].log_data[0].total := 300.0, [1068].log_data[0].time := 300.0, [1068].log_data[0].minminute := 20, [1068].log_data[0].maxminute := 20, [1068].log_data[0].valid := 1, [1068].log_data[1].valid := 1, [1068].log_data[2].valid := 1, [1068].log_data[3].valid := 1, [1068].log_data[4].valid := 1, [1068].log_data[5].valid := 1,
        [1068].log_data[6].valid := 1, [1068].log_data[7].valid := 1, [1068].log_data[8].valid := 1, [1068].log_data[9].valid := 1, [1068].log_data[10].valid := 1, [1068].log_data[11].valid := 1, [1068].log_data[12].valid := 1, [1068].log_data[13].valid := 1, [1068].log_data[14].valid := 1, [1068].log_data[15].valid := 1, [1068].log_data[16].valid := 1, [1068].log_data[17].valid := 1, [1068].log_data[18].valid := 1, [1068].log_data[19].valid := 1, [1068].time.Year := 2023, [1068].time.Month := 1, [1068].time.Day := 13, [1068].time.Hour := 9, [1068].time.Minute := 24, [1068].time.Second := 59, [1069].log_data[0].min := 1.0, [1069].log_data[0].max := 1.0, [1069].log_data[0].total := 300.0, [1069].log_data[0].time := 300.0, [1069].log_data[0].minminute := 25, [1069].log_data[0].maxminute := 25, [1069].log_data[0].valid := 1, [1069].log_data[1].valid := 1, [1069].log_data[2].valid := 1, [1069].log_data[3].valid := 1, [1069].log_data[4].valid := 1, [1069].log_data[5].valid := 1, [1069].log_data[6].valid := 1, [1069].log_data[7].valid := 1, [1069].log_data[8].valid := 1, [1069].log_data[9].valid := 1, [1069].log_data[10].valid := 1, [1069].log_data[11].valid := 1, [1069].log_data[12].valid := 1, [1069].log_data[13].valid := 1, [1069].log_data[14].valid := 1, [1069].log_data[15].valid := 1, [1069].log_data[16].valid := 1, [1069].log_data[17].valid := 1, [1069].log_data[18].valid := 1, [1069].log_data[19].valid := 1, [1069].time.Year := 2023, [1069].time.Month := 1, [1069].time.Day := 13, [1069].time.Hour := 9, [1069].time.Minute := 29, [1069].time.Second := 59, [1070].log_data[0].min := 1.0, [1070].log_data[0].max := 1.0, [1070].log_data[0].total := 300.0, [1070].log_data[0].time := 300.0, [1070].log_data[0].minminute := 30, [1070].log_data[0].maxminute := 30, [1070].log_data[0].valid := 1, [1070].log_data[1].valid := 1,
        [1070].log_data[2].valid := 1, [1070].log_data[3].valid := 1, [1070].log_data[4].valid := 1, [1070].log_data[5].valid := 1, [1070].log_data[6].valid := 1, [1070].log_data[7].valid := 1, [1070].log_data[8].valid := 1, [1070].log_data[9].valid := 1, [1070].log_data[10].valid := 1, [1070].log_data[11].valid := 1, [1070].log_data[12].valid := 1, [1070].log_data[13].valid := 1, [1070].log_data[14].valid := 1, [1070].log_data[15].valid := 1, [1070].log_data[16].valid := 1, [1070].log_data[17].valid := 1, [1070].log_data[18].valid := 1, [1070].log_data[19].valid := 1, [1070].time.Year := 2023, [1070].time.Month := 1, [1070].time.Day := 13, [1070].time.Hour := 9, [1070].time.Minute := 34, [1070].time.Second := 59, [1071].log_data[0].min := 1.0, [1071].log_data[0].max := 1.0, [1071].log_data[0].total := 300.0, [1071].log_data[0].time := 300.0, [1071].log_data[0].minminute := 35, [1071].log_data[0].maxminute := 35, [1071].log_data[0].valid := 1, [1071].log_data[1].valid := 1, [1071].log_data[2].valid := 1, [1071].log_data[3].valid := 1, [1071].log_data[4].valid := 1, [1071].log_data[5].valid := 1, [1071].log_data[6].valid := 1, [1071].log_data[7].valid := 1, [1071].log_data[8].valid := 1, [1071].log_data[9].valid := 1, [1071].log_data[10].valid := 1, [1071].log_data[11].valid := 1, [1071].log_data[12].valid := 1, [1071].log_data[13].valid := 1, [1071].log_data[14].valid := 1, [1071].log_data[15].valid := 1, [1071].log_data[16].valid := 1, [1071].log_data[17].valid := 1, [1071].log_data[18].valid := 1, [1071].log_data[19].valid := 1, [1071].time.Year := 2023, [1071].time.Month := 1, [1071].time.Day := 13, [1071].time.Hour := 9, [1071].time.Minute := 39, [1071].time.Second := 59, [1072].log_data[0].min := 1.0, [1072].log_data[0].max := 1.0, [1072].log_data[0].total := 300.0, [1072].log_data[0].time := 300.0,
        [1072].log_data[0].minminute := 40, [1072].log_data[0].maxminute := 40, [1072].log_data[0].valid := 1, [1072].log_data[1].valid := 1, [1072].log_data[2].valid := 1, [1072].log_data[3].valid := 1, [1072].log_data[4].valid := 1, [1072].log_data[5].valid := 1, [1072].log_data[6].valid := 1, [1072].log_data[7].valid := 1, [1072].log_data[8].valid := 1, [1072].log_data[9].valid := 1, [1072].log_data[10].valid := 1, [1072].log_data[11].valid := 1, [1072].log_data[12].valid := 1, [1072].log_data[13].valid := 1, [1072].log_data[14].valid := 1, [1072].log_data[15].valid := 1, [1072].log_data[16].valid := 1, [1072].log_data[17].valid := 1, [1072].log_data[18].valid := 1, [1072].log_data[19].valid := 1, [1072].time.Year := 2023, [1072].time.Month := 1, [1072].time.Day := 13, [1072].time.Hour := 9, [1072].time.Minute := 44, [1072].time.Second := 59, [1073].log_data[0].min := 1.0, [1073].log_data[0].max := 1.0, [1073].log_data[0].total := 300.0, [1073].log_data[0].time := 300.0, [1073].log_data[0].minminute := 45, [1073].log_data[0].maxminute := 45, [1073].log_data[0].valid := 1, [1073].log_data[1].valid := 1, [1073].log_data[2].valid := 1, [1073].log_data[3].valid := 1, [1073].log_data[4].valid := 1, [1073].log_data[5].valid := 1, [1073].log_data[6].valid := 1, [1073].log_data[7].valid := 1, [1073].log_data[8].valid := 1, [1073].log_data[9].valid := 1, [1073].log_data[10].valid := 1, [1073].log_data[11].valid := 1, [1073].log_data[12].valid := 1, [1073].log_data[13].valid := 1, [1073].log_data[14].valid := 1, [1073].log_data[15].valid := 1, [1073].log_data[16].valid := 1, [1073].log_data[17].valid := 1, [1073].log_data[18].valid := 1, [1073].log_data[19].valid := 1, [1073].time.Year := 2023, [1073].time.Month := 1, [1073].time.Day := 13, [1073].time.Hour := 9, [1073].time.Minute := 49, [1073].time.Second := 59,
        [1074].log_data[0].min := 1.0, [1074].log_data[0].max := 1.0, [1074].log_data[0].total := 300.0, [1074].log_data[0].time := 300.0, [1074].log_data[0].minminute := 50, [1074].log_data[0].maxminute := 50, [1074].log_data[0].valid := 1, [1074].log_data[1].valid := 1, [1074].log_data[2].valid := 1, [1074].log_data[3].valid := 1, [1074].log_data[4].valid := 1, [1074].log_data[5].valid := 1, [1074].log_data[6].valid := 1, [1074].log_data[7].valid := 1, [1074].log_data[8].valid := 1, [1074].log_data[9].valid := 1, [1074].log_data[10].valid := 1, [1074].log_data[11].valid := 1, [1074].log_data[12].valid := 1, [1074].log_data[13].valid := 1, [1074].log_data[14].valid := 1, [1074].log_data[15].valid := 1, [1074].log_data[16].valid := 1, [1074].log_data[17].valid := 1, [1074].log_data[18].valid := 1, [1074].log_data[19].valid := 1, [1074].time.Year := 2023, [1074].time.Month := 1, [1074].time.Day := 13, [1074].time.Hour := 9, [1074].time.Minute := 54, [1074].time.Second := 59, [1075].log_data[0].min := 1.0, [1075].log_data[0].max := 1.0, [1075].log_data[0].total := 300.0, [1075].log_data[0].time := 300.0, [1075].log_data[0].minminute := 55, [1075].log_data[0].maxminute := 55, [1075].log_data[0].valid := 1, [1075].log_data[1].valid := 1, [1075].log_data[2].valid := 1, [1075].log_data[3].valid := 1, [1075].log_data[4].valid := 1, [1075].log_data[5].valid := 1, [1075].log_data[6].valid := 1, [1075].log_data[7].valid := 1, [1075].log_data[8].valid := 1, [1075].log_data[9].valid := 1, [1075].log_data[10].valid := 1, [1075].log_data[11].valid := 1, [1075].log_data[12].valid := 1, [1075].log_data[13].valid := 1, [1075].log_data[14].valid := 1, [1075].log_data[15].valid := 1, [1075].log_data[16].valid := 1, [1075].log_data[17].valid := 1, [1075].log_data[18].valid := 1, [1075].log_data[19].valid := 1, [1075].time.Year := 2023, [1075].time.Month := 1,
        [1075].time.Day := 13, [1075].time.Hour := 9, [1075].time.Minute := 59, [1075].time.Second := 59, [1076].log_data[0].min := 1.0, [1076].log_data[0].max := 1.0, [1076].log_data[0].total := 300.0, [1076].log_data[0].time := 300.0, [1076].log_data[0].valid := 1, [1076].log_data[1].valid := 1, [1076].log_data[2].valid := 1, [1076].log_data[3].valid := 1, [1076].log_data[4].valid := 1, [1076].log_data[5].valid := 1, [1076].log_data[6].valid := 1, [1076].log_data[7].valid := 1, [1076].log_data[8].valid := 1, [1076].log_data[9].valid := 1, [1076].log_data[10].valid := 1, [1076].log_data[11].valid := 1, [1076].log_data[12].valid := 1, [1076].log_data[13].valid := 1, [1076].log_data[14].valid := 1, [1076].log_data[15].valid := 1, [1076].log_data[16].valid := 1, [1076].log_data[17].valid := 1, [1076].log_data[18].valid := 1, [1076].log_data[19].valid := 1, [1076].time.Year := 2023, [1076].time.Month := 1, [1076].time.Day := 13, [1076].time.Hour := 10, [1076].time.Minute := 4, [1076].time.Second := 59, [1077].log_data[0].min := 1.0, [1077].log_data[0].max := 1.0, [1077].log_data[0].total := 300.0, [1077].log_data[0].time := 300.0, [1077].log_data[0].minminute := 5, [1077].log_data[0].maxminute := 5, [1077].log_data[0].valid := 1, [1077].log_data[1].valid := 1, [1077].log_data[2].valid := 1, [1077].log_data[3].valid := 1, [1077].log_data[4].valid := 1, [1077].log_data[5].valid := 1, [1077].log_data[6].valid := 1, [1077].log_data[7].valid := 1, [1077].log_data[8].valid := 1, [1077].log_data[9].valid := 1, [1077].log_data[10].valid := 1, [1077].log_data[11].valid := 1, [1077].log_data[12].valid := 1, [1077].log_data[13].valid := 1, [1077].log_data[14].valid := 1, [1077].log_data[15].valid := 1, [1077].log_data[16].valid := 1, [1077].log_data[17].valid := 1, [1077].log_data[18].valid := 1, [1077].log_data[19].valid := 1,
        [1077].time.Year := 2023, [1077].time.Month := 1, [1077].time.Day := 13, [1077].time.Hour := 10, [1077].time.Minute := 9, [1077].time.Second := 59, [1078].log_data[0].min := 1.0, [1078].log_data[0].max := 1.0, [1078].log_data[0].total := 300.0, [1078].log_data[0].time := 300.0, [1078].log_data[0].minminute := 10, [1078].log_data[0].maxminute := 10, [1078].log_data[0].valid := 1, [1078].log_data[1].valid := 1, [1078].log_data[2].valid := 1, [1078].log_data[3].valid := 1, [1078].log_data[4].valid := 1, [1078].log_data[5].valid := 1, [1078].log_data[6].valid := 1, [1078].log_data[7].valid := 1, [1078].log_data[8].valid := 1, [1078].log_data[9].valid := 1, [1078].log_data[10].valid := 1, [1078].log_data[11].valid := 1, [1078].log_data[12].valid := 1, [1078].log_data[13].valid := 1, [1078].log_data[14].valid := 1, [1078].log_data[15].valid := 1, [1078].log_data[16].valid := 1, [1078].log_data[17].valid := 1, [1078].log_data[18].valid := 1, [1078].log_data[19].valid := 1, [1078].time.Year := 2023, [1078].time.Month := 1, [1078].time.Day := 13, [1078].time.Hour := 10, [1078].time.Minute := 14, [1078].time.Second := 59, [1079].log_data[0].min := 1.0, [1079].log_data[0].max := 1.0, [1079].log_data[0].total := 300.0, [1079].log_data[0].time := 300.0, [1079].log_data[0].minminute := 15, [1079].log_data[0].maxminute := 15, [1079].log_data[0].valid := 1, [1079].log_data[1].valid := 1, [1079].log_data[2].valid := 1, [1079].log_data[3].valid := 1, [1079].log_data[4].valid := 1, [1079].log_data[5].valid := 1, [1079].log_data[6].valid := 1, [1079].log_data[7].valid := 1, [1079].log_data[8].valid := 1, [1079].log_data[9].valid := 1, [1079].log_data[10].valid := 1, [1079].log_data[11].valid := 1, [1079].log_data[12].valid := 1, [1079].log_data[13].valid := 1, [1079].log_data[14].valid := 1, [1079].log_data[15].valid := 1,
        [1079].log_data[16].valid := 1, [1079].log_data[17].valid := 1, [1079].log_data[18].valid := 1, [1079].log_data[19].valid := 1, [1079].time.Year := 2023, [1079].time.Month := 1, [1079].time.Day := 13, [1079].time.Hour := 10, [1079].time.Minute := 19, [1079].time.Second := 59, [1080].log_data[0].min := 1.0, [1080].log_data[0].max := 1.0, [1080].log_data[0].total := 300.0, [1080].log_data[0].time := 300.0, [1080].log_data[0].minminute := 20, [1080].log_data[0].maxminute := 20, [1080].log_data[0].valid := 1, [1080].log_data[1].valid := 1, [1080].log_data[2].valid := 1, [1080].log_data[3].valid := 1, [1080].log_data[4].valid := 1, [1080].log_data[5].valid := 1, [1080].log_data[6].valid := 1, [1080].log_data[7].valid := 1, [1080].log_data[8].valid := 1, [1080].log_data[9].valid := 1, [1080].log_data[10].valid := 1, [1080].log_data[11].valid := 1, [1080].log_data[12].valid := 1, [1080].log_data[13].valid := 1, [1080].log_data[14].valid := 1, [1080].log_data[15].valid := 1, [1080].log_data[16].valid := 1, [1080].log_data[17].valid := 1, [1080].log_data[18].valid := 1, [1080].log_data[19].valid := 1, [1080].time.Year := 2023, [1080].time.Month := 1, [1080].time.Day := 13, [1080].time.Hour := 10, [1080].time.Minute := 24, [1080].time.Second := 59, [1081].log_data[0].min := 1.0, [1081].log_data[0].max := 1.0, [1081].log_data[0].total := 300.0, [1081].log_data[0].time := 300.0, [1081].log_data[0].minminute := 25, [1081].log_data[0].maxminute := 25, [1081].log_data[0].valid := 1, [1081].log_data[1].valid := 1, [1081].log_data[2].valid := 1, [1081].log_data[3].valid := 1, [1081].log_data[4].valid := 1, [1081].log_data[5].valid := 1, [1081].log_data[6].valid := 1, [1081].log_data[7].valid := 1, [1081].log_data[8].valid := 1, [1081].log_data[9].valid := 1, [1081].log_data[10].valid := 1, [1081].log_data[11].valid := 1,
        [1081].log_data[12].valid := 1, [1081].log_data[13].valid := 1, [1081].log_data[14].valid := 1, [1081].log_data[15].valid := 1, [1081].log_data[16].valid := 1, [1081].log_data[17].valid := 1, [1081].log_data[18].valid := 1, [1081].log_data[19].valid := 1, [1081].time.Year := 2023, [1081].time.Month := 1, [1081].time.Day := 13, [1081].time.Hour := 10, [1081].time.Minute := 29, [1081].time.Second := 59, [1082].log_data[0].min := 1.0, [1082].log_data[0].max := 1.0, [1082].log_data[0].total := 300.0, [1082].log_data[0].time := 300.0, [1082].log_data[0].minminute := 30, [1082].log_data[0].maxminute := 30, [1082].log_data[0].valid := 1, [1082].log_data[1].valid := 1, [1082].log_data[2].valid := 1, [1082].log_data[3].valid := 1, [1082].log_data[4].valid := 1, [1082].log_data[5].valid := 1, [1082].log_data[6].valid := 1, [1082].log_data[7].valid := 1, [1082].log_data[8].valid := 1, [1082].log_data[9].valid := 1, [1082].log_data[10].valid := 1, [1082].log_data[11].valid := 1, [1082].log_data[12].valid := 1, [1082].log_data[13].valid := 1, [1082].log_data[14].valid := 1, [1082].log_data[15].valid := 1, [1082].log_data[16].valid := 1, [1082].log_data[17].valid := 1, [1082].log_data[18].valid := 1, [1082].log_data[19].valid := 1, [1082].time.Year := 2023, [1082].time.Month := 1, [1082].time.Day := 13, [1082].time.Hour := 10, [1082].time.Minute := 34, [1082].time.Second := 59, [1083].log_data[0].min := 1.0, [1083].log_data[0].max := 1.0, [1083].log_data[0].total := 300.0, [1083].log_data[0].time := 300.0, [1083].log_data[0].minminute := 35, [1083].log_data[0].maxminute := 35, [1083].log_data[0].valid := 1, [1083].log_data[1].valid := 1, [1083].log_data[2].valid := 1, [1083].log_data[3].valid := 1, [1083].log_data[4].valid := 1, [1083].log_data[5].valid := 1, [1083].log_data[6].valid := 1, [1083].log_data[7].valid := 1,
        [1083].log_data[8].valid := 1, [1083].log_data[9].valid := 1, [1083].log_data[10].valid := 1, [1083].log_data[11].valid := 1, [1083].log_data[12].valid := 1, [1083].log_data[13].valid := 1, [1083].log_data[14].valid := 1, [1083].log_data[15].valid := 1, [1083].log_data[16].valid := 1, [1083].log_data[17].valid := 1, [1083].log_data[18].valid := 1, [1083].log_data[19].valid := 1, [1083].time.Year := 2023, [1083].time.Month := 1, [1083].time.Day := 13, [1083].time.Hour := 10, [1083].time.Minute := 39, [1083].time.Second := 59, [1084].log_data[0].min := 1.0, [1084].log_data[0].max := 1.0, [1084].log_data[0].total := 300.0, [1084].log_data[0].time := 300.0, [1084].log_data[0].minminute := 40, [1084].log_data[0].maxminute := 40, [1084].log_data[0].valid := 1, [1084].log_data[1].valid := 1, [1084].log_data[2].valid := 1, [1084].log_data[3].valid := 1, [1084].log_data[4].valid := 1, [1084].log_data[5].valid := 1, [1084].log_data[6].valid := 1, [1084].log_data[7].valid := 1, [1084].log_data[8].valid := 1, [1084].log_data[9].valid := 1, [1084].log_data[10].valid := 1, [1084].log_data[11].valid := 1, [1084].log_data[12].valid := 1, [1084].log_data[13].valid := 1, [1084].log_data[14].valid := 1, [1084].log_data[15].valid := 1, [1084].log_data[16].valid := 1, [1084].log_data[17].valid := 1, [1084].log_data[18].valid := 1, [1084].log_data[19].valid := 1, [1084].time.Year := 2023, [1084].time.Month := 1, [1084].time.Day := 13, [1084].time.Hour := 10, [1084].time.Minute := 44, [1084].time.Second := 59, [1085].log_data[0].min := 1.0, [1085].log_data[0].max := 1.0, [1085].log_data[0].total := 300.0, [1085].log_data[0].time := 300.0, [1085].log_data[0].minminute := 45, [1085].log_data[0].maxminute := 45, [1085].log_data[0].valid := 1, [1085].log_data[1].valid := 1, [1085].log_data[2].valid := 1, [1085].log_data[3].valid := 1,
        [1085].log_data[4].valid := 1, [1085].log_data[5].valid := 1, [1085].log_data[6].valid := 1, [1085].log_data[7].valid := 1, [1085].log_data[8].valid := 1, [1085].log_data[9].valid := 1, [1085].log_data[10].valid := 1, [1085].log_data[11].valid := 1, [1085].log_data[12].valid := 1, [1085].log_data[13].valid := 1, [1085].log_data[14].valid := 1, [1085].log_data[15].valid := 1, [1085].log_data[16].valid := 1, [1085].log_data[17].valid := 1, [1085].log_data[18].valid := 1, [1085].log_data[19].valid := 1, [1085].time.Year := 2023, [1085].time.Month := 1, [1085].time.Day := 13, [1085].time.Hour := 10, [1085].time.Minute := 49, [1085].time.Second := 59, [1086].log_data[0].min := 1.0, [1086].log_data[0].max := 1.0, [1086].log_data[0].total := 300.0, [1086].log_data[0].time := 300.0, [1086].log_data[0].minminute := 50, [1086].log_data[0].maxminute := 50, [1086].log_data[0].valid := 1, [1086].log_data[1].valid := 1, [1086].log_data[2].valid := 1, [1086].log_data[3].valid := 1, [1086].log_data[4].valid := 1, [1086].log_data[5].valid := 1, [1086].log_data[6].valid := 1, [1086].log_data[7].valid := 1, [1086].log_data[8].valid := 1, [1086].log_data[9].valid := 1, [1086].log_data[10].valid := 1, [1086].log_data[11].valid := 1, [1086].log_data[12].valid := 1, [1086].log_data[13].valid := 1, [1086].log_data[14].valid := 1, [1086].log_data[15].valid := 1, [1086].log_data[16].valid := 1, [1086].log_data[17].valid := 1, [1086].log_data[18].valid := 1, [1086].log_data[19].valid := 1, [1086].time.Year := 2023, [1086].time.Month := 1, [1086].time.Day := 13, [1086].time.Hour := 10, [1086].time.Minute := 54, [1086].time.Second := 59, [1087].log_data[0].min := 1.0, [1087].log_data[0].max := 1.0, [1087].log_data[0].total := 300.0, [1087].log_data[0].time := 300.0, [1087].log_data[0].minminute := 55, [1087].log_data[0].maxminute := 55,
        [1087].log_data[0].valid := 1, [1087].log_data[1].valid := 1, [1087].log_data[2].valid := 1, [1087].log_data[3].valid := 1, [1087].log_data[4].valid := 1, [1087].log_data[5].valid := 1, [1087].log_data[6].valid := 1, [1087].log_data[7].valid := 1, [1087].log_data[8].valid := 1, [1087].log_data[9].valid := 1, [1087].log_data[10].valid := 1, [1087].log_data[11].valid := 1, [1087].log_data[12].valid := 1, [1087].log_data[13].valid := 1, [1087].log_data[14].valid := 1, [1087].log_data[15].valid := 1, [1087].log_data[16].valid := 1, [1087].log_data[17].valid := 1, [1087].log_data[18].valid := 1, [1087].log_data[19].valid := 1, [1087].time.Year := 2023, [1087].time.Month := 1, [1087].time.Day := 13, [1087].time.Hour := 10, [1087].time.Minute := 59, [1087].time.Second := 59, [1088].log_data[0].min := 1.0, [1088].log_data[0].max := 1.0, [1088].log_data[0].total := 300.0, [1088].log_data[0].time := 300.0, [1088].log_data[0].valid := 1, [1088].log_data[1].valid := 1, [1088].log_data[2].valid := 1, [1088].log_data[3].valid := 1, [1088].log_data[4].valid := 1, [1088].log_data[5].valid := 1, [1088].log_data[6].valid := 1, [1088].log_data[7].valid := 1, [1088].log_data[8].valid := 1, [1088].log_data[9].valid := 1, [1088].log_data[10].valid := 1, [1088].log_data[11].valid := 1, [1088].log_data[12].valid := 1, [1088].log_data[13].valid := 1, [1088].log_data[14].valid := 1, [1088].log_data[15].valid := 1, [1088].log_data[16].valid := 1, [1088].log_data[17].valid := 1, [1088].log_data[18].valid := 1, [1088].log_data[19].valid := 1, [1088].time.Year := 2023, [1088].time.Month := 1, [1088].time.Day := 13, [1088].time.Hour := 11, [1088].time.Minute := 4, [1088].time.Second := 59, [1089].log_data[0].min := 1.0, [1089].log_data[0].max := 1.0, [1089].log_data[0].total := 300.0, [1089].log_data[0].time := 300.0,
        [1089].log_data[0].minminute := 5, [1089].log_data[0].maxminute := 5, [1089].log_data[0].valid := 1, [1089].log_data[1].valid := 1, [1089].log_data[2].valid := 1, [1089].log_data[3].valid := 1, [1089].log_data[4].valid := 1, [1089].log_data[5].valid := 1, [1089].log_data[6].valid := 1, [1089].log_data[7].valid := 1, [1089].log_data[8].valid := 1, [1089].log_data[9].valid := 1, [1089].log_data[10].valid := 1, [1089].log_data[11].valid := 1, [1089].log_data[12].valid := 1, [1089].log_data[13].valid := 1, [1089].log_data[14].valid := 1, [1089].log_data[15].valid := 1, [1089].log_data[16].valid := 1, [1089].log_data[17].valid := 1, [1089].log_data[18].valid := 1, [1089].log_data[19].valid := 1, [1089].time.Year := 2023, [1089].time.Month := 1, [1089].time.Day := 13, [1089].time.Hour := 11, [1089].time.Minute := 9, [1089].time.Second := 59, [1090].log_data[0].min := 1.0, [1090].log_data[0].max := 1.0, [1090].log_data[0].total := 300.0, [1090].log_data[0].time := 300.0, [1090].log_data[0].minminute := 10, [1090].log_data[0].maxminute := 10, [1090].log_data[0].valid := 1, [1090].log_data[1].valid := 1, [1090].log_data[2].valid := 1, [1090].log_data[3].valid := 1, [1090].log_data[4].valid := 1, [1090].log_data[5].valid := 1, [1090].log_data[6].valid := 1, [1090].log_data[7].valid := 1, [1090].log_data[8].valid := 1, [1090].log_data[9].valid := 1, [1090].log_data[10].valid := 1, [1090].log_data[11].valid := 1, [1090].log_data[12].valid := 1, [1090].log_data[13].valid := 1, [1090].log_data[14].valid := 1, [1090].log_data[15].valid := 1, [1090].log_data[16].valid := 1, [1090].log_data[17].valid := 1, [1090].log_data[18].valid := 1, [1090].log_data[19].valid := 1, [1090].time.Year := 2023, [1090].time.Month := 1, [1090].time.Day := 13, [1090].time.Hour := 11, [1090].time.Minute := 14, [1090].time.Second := 59,
        [1091].log_data[0].min := 1.0, [1091].log_data[0].max := 1.0, [1091].log_data[0].total := 300.0, [1091].log_data[0].time := 300.0, [1091].log_data[0].minminute := 15, [1091].log_data[0].maxminute := 15, [1091].log_data[0].valid := 1, [1091].log_data[1].valid := 1, [1091].log_data[2].valid := 1, [1091].log_data[3].valid := 1, [1091].log_data[4].valid := 1, [1091].log_data[5].valid := 1, [1091].log_data[6].valid := 1, [1091].log_data[7].valid := 1, [1091].log_data[8].valid := 1, [1091].log_data[9].valid := 1, [1091].log_data[10].valid := 1, [1091].log_data[11].valid := 1, [1091].log_data[12].valid := 1, [1091].log_data[13].valid := 1, [1091].log_data[14].valid := 1, [1091].log_data[15].valid := 1, [1091].log_data[16].valid := 1, [1091].log_data[17].valid := 1, [1091].log_data[18].valid := 1, [1091].log_data[19].valid := 1, [1091].time.Year := 2023, [1091].time.Month := 1, [1091].time.Day := 13, [1091].time.Hour := 11, [1091].time.Minute := 19, [1091].time.Second := 59, [1092].log_data[0].min := 1.0, [1092].log_data[0].max := 1.0, [1092].log_data[0].total := 300.0, [1092].log_data[0].time := 300.0, [1092].log_data[0].minminute := 20, [1092].log_data[0].maxminute := 20, [1092].log_data[0].valid := 1, [1092].log_data[1].valid := 1, [1092].log_data[2].valid := 1, [1092].log_data[3].valid := 1, [1092].log_data[4].valid := 1, [1092].log_data[5].valid := 1, [1092].log_data[6].valid := 1, [1092].log_data[7].valid := 1, [1092].log_data[8].valid := 1, [1092].log_data[9].valid := 1, [1092].log_data[10].valid := 1, [1092].log_data[11].valid := 1, [1092].log_data[12].valid := 1, [1092].log_data[13].valid := 1, [1092].log_data[14].valid := 1, [1092].log_data[15].valid := 1, [1092].log_data[16].valid := 1, [1092].log_data[17].valid := 1, [1092].log_data[18].valid := 1, [1092].log_data[19].valid := 1, [1092].time.Year := 2023, [1092].time.Month := 1,
        [1092].time.Day := 13, [1092].time.Hour := 11, [1092].time.Minute := 24, [1092].time.Second := 59, [1093].log_data[0].min := 1.0, [1093].log_data[0].max := 1.0, [1093].log_data[0].total := 300.0, [1093].log_data[0].time := 300.0, [1093].log_data[0].minminute := 25, [1093].log_data[0].maxminute := 25, [1093].log_data[0].valid := 1, [1093].log_data[1].valid := 1, [1093].log_data[2].valid := 1, [1093].log_data[3].valid := 1, [1093].log_data[4].valid := 1, [1093].log_data[5].valid := 1, [1093].log_data[6].valid := 1, [1093].log_data[7].valid := 1, [1093].log_data[8].valid := 1, [1093].log_data[9].valid := 1, [1093].log_data[10].valid := 1, [1093].log_data[11].valid := 1, [1093].log_data[12].valid := 1, [1093].log_data[13].valid := 1, [1093].log_data[14].valid := 1, [1093].log_data[15].valid := 1, [1093].log_data[16].valid := 1, [1093].log_data[17].valid := 1, [1093].log_data[18].valid := 1, [1093].log_data[19].valid := 1, [1093].time.Year := 2023, [1093].time.Month := 1, [1093].time.Day := 13, [1093].time.Hour := 11, [1093].time.Minute := 29, [1093].time.Second := 59, [1094].log_data[0].min := 1.0, [1094].log_data[0].max := 1.0, [1094].log_data[0].total := 300.0, [1094].log_data[0].time := 300.0, [1094].log_data[0].minminute := 30, [1094].log_data[0].maxminute := 30, [1094].log_data[0].valid := 1, [1094].log_data[1].valid := 1, [1094].log_data[2].valid := 1, [1094].log_data[3].valid := 1, [1094].log_data[4].valid := 1, [1094].log_data[5].valid := 1, [1094].log_data[6].valid := 1, [1094].log_data[7].valid := 1, [1094].log_data[8].valid := 1, [1094].log_data[9].valid := 1, [1094].log_data[10].valid := 1, [1094].log_data[11].valid := 1, [1094].log_data[12].valid := 1, [1094].log_data[13].valid := 1, [1094].log_data[14].valid := 1, [1094].log_data[15].valid := 1, [1094].log_data[16].valid := 1, [1094].log_data[17].valid := 1,
        [1094].log_data[18].valid := 1, [1094].log_data[19].valid := 1, [1094].time.Year := 2023, [1094].time.Month := 1, [1094].time.Day := 13, [1094].time.Hour := 11, [1094].time.Minute := 34, [1094].time.Second := 59, [1095].log_data[0].min := 1.0, [1095].log_data[0].max := 1.0, [1095].log_data[0].total := 300.0, [1095].log_data[0].time := 300.0, [1095].log_data[0].minminute := 35, [1095].log_data[0].maxminute := 35, [1095].log_data[0].valid := 1, [1095].log_data[1].valid := 1, [1095].log_data[2].valid := 1, [1095].log_data[3].valid := 1, [1095].log_data[4].valid := 1, [1095].log_data[5].valid := 1, [1095].log_data[6].valid := 1, [1095].log_data[7].valid := 1, [1095].log_data[8].valid := 1, [1095].log_data[9].valid := 1, [1095].log_data[10].valid := 1, [1095].log_data[11].valid := 1, [1095].log_data[12].valid := 1, [1095].log_data[13].valid := 1, [1095].log_data[14].valid := 1, [1095].log_data[15].valid := 1, [1095].log_data[16].valid := 1, [1095].log_data[17].valid := 1, [1095].log_data[18].valid := 1, [1095].log_data[19].valid := 1, [1095].time.Year := 2023, [1095].time.Month := 1, [1095].time.Day := 13, [1095].time.Hour := 11, [1095].time.Minute := 39, [1095].time.Second := 59, [1096].log_data[0].min := 1.0, [1096].log_data[0].max := 1.0, [1096].log_data[0].total := 300.0, [1096].log_data[0].time := 300.0, [1096].log_data[0].minminute := 40, [1096].log_data[0].maxminute := 40, [1096].log_data[0].valid := 1, [1096].log_data[1].valid := 1, [1096].log_data[2].valid := 1, [1096].log_data[3].valid := 1, [1096].log_data[4].valid := 1, [1096].log_data[5].valid := 1, [1096].log_data[6].valid := 1, [1096].log_data[7].valid := 1, [1096].log_data[8].valid := 1, [1096].log_data[9].valid := 1, [1096].log_data[10].valid := 1, [1096].log_data[11].valid := 1, [1096].log_data[12].valid := 1, [1096].log_data[13].valid := 1,
